LIN {X 0,Y 409.428,Z 527.797,A -85,B 0,C 180,E1 19478.338,E2 19478.338} C_VEL
LIN {X 0,Y 409.412,Z 527.774,A -85,B 0,C 180,E1 19474.343,E2 19474.343} C_VEL
LIN {X 0,Y 409.395,Z 527.8,A -85,B 0,C 180,E1 19470.531,E2 19470.531} C_VEL
LIN {X 0,Y 409.376,Z 527.779,A -85,B 0,C 180,E1 19466.862,E2 19466.862} C_VEL
LIN {X 0,Y 409.379,Z 527.798,A -85,B 0,C 180,E1 19462.967,E2 19462.967} C_VEL
LIN {X 0,Y 409.396,Z 527.782,A -85,B 0,C 180,E1 19459.251,E2 19459.251} C_VEL
LIN {X 0,Y 409.422,Z 527.785,A -85,B 0,C 180,E1 19455.438,E2 19455.438} C_VEL
LIN {X 0,Y 409.43,Z 527.788,A -85,B 0,C 180,E1 19451.552,E2 19451.552} C_VEL
LIN {X 0,Y 409.424,Z 527.77,A -85,B 0,C 180,E1 19447.578,E2 19447.578} C_VEL
LIN {X 0,Y 409.403,Z 527.799,A -85,B 0,C 180,E1 19443.781,E2 19443.781} C_VEL
LIN {X 0,Y 409.386,Z 527.767,A -85,B 0,C 180,E1 19440,E2 19440} C_VEL
LIN {X 0,Y 409.39,Z 527.799,A -85,B 0,C 180,E1 19436.079,E2 19436.079} C_VEL
LIN {X 0,Y 409.392,Z 527.773,A -85,B 0,C 180,E1 19432.139,E2 19432.139} C_VEL
LIN {X 0,Y 409.409,Z 527.797,A -85,B 0,C 180,E1 19428.305,E2 19428.305} C_VEL
LIN {X 0,Y 409.427,Z 527.78,A -85,B 0,C 180,E1 19424.417,E2 19424.417} C_VEL
LIN {X 0,Y 409.438,Z 527.787,A -85,B 0,C 180,E1 19420.488,E2 19420.488} C_VEL
LIN {X 0,Y 409.444,Z 527.796,A -85,B 0,C 180,E1 19416.544,E2 19416.544} C_VEL
LIN {X 0,Y 409.427,Z 527.783,A -85,B 0,C 180,E1 19412.67,E2 19412.67} C_VEL
LIN {X 0,Y 409.405,Z 527.789,A -85,B 0,C 180,E1 19408.982,E2 19408.982} C_VEL
LIN {X 0,Y 409.402,Z 527.793,A -85,B 0,C 180,E1 19405.14,E2 19405.14} C_VEL
LIN {X 0,Y 409.412,Z 527.79,A -85,B 0,C 180,E1 19401.303,E2 19401.303} C_VEL
LIN {X 0,Y 409.43,Z 527.79,A -85,B 0,C 180,E1 19397.516,E2 19397.516} C_VEL
LIN {X 0,Y 409.443,Z 527.799,A -85,B 0,C 180,E1 19393.711,E2 19393.711} C_VEL
LIN {X 0,Y 409.472,Z 528.088,A -85,B 0,C 180,E1 19392.071,E2 19392.071} C_VEL
LIN {X 0,Y 417.086,Z 549.044,A -85,B 0,C 180,E1 19388.821,E2 19388.821} C_VEL
LIN {X 0,Y 424.699,Z 571.518,A -85,B 0,C 180,E1 19385.686,E2 19385.686} C_VEL
LIN {X 0,Y 421.199,Z 607.599,A -85,B 0,C 180,E1 19382.122,E2 19382.122} C_VEL
LIN {X 0,Y 420.389,Z 616.971,A -85,B 0,C 180,E1 19381.23,E2 19381.23} C_VEL
LIN {X 0,Y 423.028,Z 641.822,A -85,B 0,C 180,E1 19380.601,E2 19380.601} C_VEL
LIN {X 0,Y 420.192,Z 815.687,A -85,B 0,C 180,E1 19377.631,E2 19377.631} C_VEL
LIN {X 0,Y 419.282,Z 834.324,A -85,B 0,C 180,E1 19377.076,E2 19377.076} C_VEL
LIN {X 0,Y 418.101,Z 852.187,A -85,B 0,C 180,E1 19376.296,E2 19376.296} C_VEL
LIN {X 0,Y 416.736,Z 869.515,A -85,B 0,C 180,E1 19375.281,E2 19375.281} C_VEL
LIN {X 0,Y 415.229,Z 886.464,A -85,B 0,C 180,E1 19374.013,E2 19374.013} C_VEL
LIN {X 0,Y 413.683,Z 902.434,A -85,B 0,C 180,E1 19372.525,E2 19372.525} C_VEL
LIN {X 0,Y 412.253,Z 917.439,A -85,B 0,C 180,E1 19370.813,E2 19370.813} C_VEL
LIN {X 0,Y 410.942,Z 931.411,A -85,B 0,C 180,E1 19368.881,E2 19368.881} C_VEL
LIN {X 0,Y 409.865,Z 944.229,A -85,B 0,C 180,E1 19366.73,E2 19366.73} C_VEL
LIN {X 0,Y 409.104,Z 955.381,A -85,B 0,C 180,E1 19364.436,E2 19364.436} C_VEL
LIN {X 0,Y 408.664,Z 964.433,A -85,B 0,C 180,E1 19362.147,E2 19362.147} C_VEL
LIN {X 0,Y 408.487,Z 972.044,A -85,B 0,C 180,E1 19359.724,E2 19359.724} C_VEL
LIN {X 0,Y 408.488,Z 977.818,A -85,B 0,C 180,E1 19357.314,E2 19357.314} C_VEL
LIN {X 0,Y 408.596,Z 981.892,A -85,B 0,C 180,E1 19354.915,E2 19354.915} C_VEL
LIN {X 0,Y 408.712,Z 984.339,A -85,B 0,C 180,E1 19352.525,E2 19352.525} C_VEL
LIN {X 0,Y 408.779,Z 985.198,A -85,B 0,C 180,E1 19350.002,E2 19350.002} C_VEL
LIN {X 0,Y 408.718,Z 984.298,A -85,B 0,C 180,E1 19347.478,E2 19347.478} C_VEL
LIN {X 0,Y 408.599,Z 981.642,A -85,B 0,C 180,E1 19344.948,E2 19344.948} C_VEL
LIN {X 0,Y 408.483,Z 977.183,A -85,B 0,C 180,E1 19342.407,E2 19342.407} C_VEL
LIN {X 0,Y 408.507,Z 970.81,A -85,B 0,C 180,E1 19339.853,E2 19339.853} C_VEL
LIN {X 0,Y 408.719,Z 962.882,A -85,B 0,C 180,E1 19337.428,E2 19337.428} C_VEL
LIN {X 0,Y 409.259,Z 952.866,A -85,B 0,C 180,E1 19334.994,E2 19334.994} C_VEL
LIN {X 0,Y 410.046,Z 942.036,A -85,B 0,C 180,E1 19332.843,E2 19332.843} C_VEL
LIN {X 0,Y 411.163,Z 929.405,A -85,B 0,C 180,E1 19330.766,E2 19330.766} C_VEL
LIN {X 0,Y 412.611,Z 914.663,A -85,B 0,C 180,E1 19328.764,E2 19328.764} C_VEL
LIN {X 0,Y 414.144,Z 899.377,A -85,B 0,C 180,E1 19327.055,E2 19327.055} C_VEL
LIN {X 0,Y 415.73,Z 883.929,A -85,B 0,C 180,E1 19325.644,E2 19325.644} C_VEL
LIN {X 0,Y 417.307,Z 866.913,A -85,B 0,C 180,E1 19324.388,E2 19324.388} C_VEL
LIN {X 0,Y 418.791,Z 849.197,A -85,B 0,C 180,E1 19323.373,E2 19323.373} C_VEL
LIN {X 0,Y 420.069,Z 830.603,A -85,B 0,C 180,E1 19322.594,E2 19322.594} C_VEL
LIN {X 0,Y 420.944,Z 811.694,A -85,B 0,C 180,E1 19322.072,E2 19322.072} C_VEL
LIN {X 0,Y 423.821,Z 639.08,A -85,B 0,C 180,E1 19319.074,E2 19319.074} C_VEL
LIN {X 0,Y 421.333,Z 617.013,A -85,B 0,C 180,E1 19318.434,E2 19318.434} C_VEL
LIN {X 0,Y 426.266,Z 573.613,A -85,B 0,C 180,E1 19314.039,E2 19314.039} C_VEL
LIN {X 0,Y 420.863,Z 557.04,A -85,B 0,C 180,E1 19311.511,E2 19311.511} C_VEL
LIN {X 0,Y 415.095,Z 541.83,A -85,B 0,C 180,E1 19308.89,E2 19308.89} C_VEL
LIN {X 0,Y 410.413,Z 530.778,A -85,B 0,C 180,E1 19306.755,E2 19306.755} C_VEL
LIN {X 0,Y 409.458,Z 527.95,A -85,B 0,C 180,E1 19306.13,E2 19306.13} C_VEL
LIN {X 0,Y 409.44,Z 527.788,A -85,B 0,C 180,E1 19302.187,E2 19302.187} C_VEL
LIN {X 0,Y 409.429,Z 527.787,A -85,B 0,C 180,E1 19298.337,E2 19298.337} C_VEL
LIN {X 0,Y 409.403,Z 527.796,A -85,B 0,C 180,E1 19294.513,E2 19294.513} C_VEL
LIN {X 0,Y 409.388,Z 527.799,A -85,B 0,C 180,E1 19290.693,E2 19290.693} C_VEL
LIN {X 0,Y 409.38,Z 527.798,A -85,B 0,C 180,E1 19286.862,E2 19286.862} C_VEL
LIN {X 0,Y 409.381,Z 527.791,A -85,B 0,C 180,E1 19282.977,E2 19282.977} C_VEL
LIN {X 0,Y 409.397,Z 527.783,A -85,B 0,C 180,E1 19279.251,E2 19279.251} C_VEL
LIN {X 0,Y 409.419,Z 527.784,A -85,B 0,C 180,E1 19275.438,E2 19275.438} C_VEL
LIN {X 0,Y 409.404,Z 527.801,A -85,B 0,C 180,E1 19271.552,E2 19271.552} C_VEL
LIN {X 0,Y 409.383,Z 527.799,A -85,B 0,C 180,E1 19267.72,E2 19267.72} C_VEL
LIN {X 0,Y 409.37,Z 527.787,A -85,B 0,C 180,E1 19263.921,E2 19263.921} C_VEL
LIN {X 0,Y 409.371,Z 527.786,A -85,B 0,C 180,E1 19260.14,E2 19260.14} C_VEL
LIN {X 0,Y 409.386,Z 527.796,A -85,B 0,C 180,E1 19256.359,E2 19256.359} C_VEL
LIN {X 0,Y 409.414,Z 527.799,A -85,B 0,C 180,E1 19252.563,E2 19252.563} C_VEL
LIN {X 0,Y 409.432,Z 527.798,A -85,B 0,C 180,E1 19248.734,E2 19248.734} C_VEL
LIN {X 0,Y 409.431,Z 527.795,A -85,B 0,C 180,E1 19244.852,E2 19244.852} C_VEL
LIN {X 0,Y 409.412,Z 527.798,A -85,B 0,C 180,E1 19241.046,E2 19241.046} C_VEL
LIN {X 0,Y 409.4,Z 527.803,A -85,B 0,C 180,E1 19237.301,E2 19237.301} C_VEL
LIN {X 0,Y 409.402,Z 527.794,A -85,B 0,C 180,E1 19233.349,E2 19233.349} C_VEL
LIN {X 0,Y 409.414,Z 527.839,A -85,B 0,C 180,E1 19229.471,E2 19229.471} C_VEL
LIN {X 0,Y 409.537,Z 528.542,A -85,B 0,C 180,E1 19229.156,E2 19229.156} C_VEL
LIN {X 0,Y 413.799,Z 540.293,A -85,B 0,C 180,E1 19226.404,E2 19226.404} C_VEL
LIN {X 0,Y 418.13,Z 554.109,A -85,B 0,C 180,E1 19223.453,E2 19223.453} C_VEL
LIN {X 0,Y 421.697,Z 567.85,A -85,B 0,C 180,E1 19220.767,E2 19220.767} C_VEL
LIN {X 0,Y 418.78,Z 594.647,A -85,B 0,C 180,E1 19216.728,E2 19216.728} C_VEL
LIN {X 0,Y 416.121,Z 622.884,A -85,B 0,C 180,E1 19212.555,E2 19212.555} C_VEL
LIN {X 0,Y 415.538,Z 630.261,A -85,B 0,C 180,E1 19211.502,E2 19211.502} C_VEL
LIN {X 0,Y 416.961,Z 637.693,A -85,B 0,C 180,E1 19211.191,E2 19211.191} C_VEL
LIN {X 0,Y 420.359,Z 656.969,A -85,B 0,C 180,E1 19210.559,E2 19210.559} C_VEL
LIN {X 0,Y 418.283,Z 753.864,A -85,B 0,C 180,E1 19208.726,E2 19208.726} C_VEL
LIN {X 0,Y 417.743,Z 769.981,A -85,B 0,C 180,E1 19208.156,E2 19208.156} C_VEL
LIN {X 0,Y 416.97,Z 784.418,A -85,B 0,C 180,E1 19207.391,E2 19207.391} C_VEL
LIN {X 0,Y 415.919,Z 799,A -85,B 0,C 180,E1 19206.335,E2 19206.335} C_VEL
LIN {X 0,Y 414.729,Z 811.961,A -85,B 0,C 180,E1 19205.094,E2 19205.094} C_VEL
LIN {X 0,Y 413.625,Z 823.119,A -85,B 0,C 180,E1 19203.741,E2 19203.741} C_VEL
LIN {X 0,Y 412.428,Z 833.983,A -85,B 0,C 180,E1 19202.063,E2 19202.063} C_VEL
LIN {X 0,Y 411.435,Z 842.658,A -85,B 0,C 180,E1 19200.358,E2 19200.358} C_VEL
LIN {X 0,Y 410.535,Z 850.51,A -85,B 0,C 180,E1 19198.35,E2 19198.35} C_VEL
LIN {X 0,Y 409.905,Z 856.206,A -85,B 0,C 180,E1 19196.351,E2 19196.351} C_VEL
LIN {X 0,Y 409.471,Z 860.386,A -85,B 0,C 180,E1 19194.215,E2 19194.215} C_VEL
LIN {X 0,Y 409.207,Z 862.789,A -85,B 0,C 180,E1 19191.949,E2 19191.949} C_VEL
LIN {X 0,Y 409.115,Z 863.297,A -85,B 0,C 180,E1 19189.792,E2 19189.792} C_VEL
LIN {X 0,Y 409.173,Z 861.968,A -85,B 0,C 180,E1 19187.488,E2 19187.488} C_VEL
LIN {X 0,Y 409.177,Z 861.878,A -85,B 0,C 180,E1 19187.409,E2 19187.409} C_VEL
LIN {X 0,Y 408.267,Z 860.683,A -85,B 0,C 180,E1 19186.342,E2 19186.342} C_VEL
LIN {X 0,Y 404.279,Z 858.032,A -85,B 0,C 180,E1 19184.487,E2 19184.487} C_VEL
LIN {X 0,Y 402.202,Z 855.385,A -85,B 0,C 180,E1 19183.225,E2 19183.225} C_VEL
LIN {X 0,Y 402.01,Z 853.771,A -85,B 0,C 180,E1 19182.633,E2 19182.633} C_VEL
LIN {X 0,Y 402.625,Z 847.266,A -85,B 0,C 180,E1 19180.731,E2 19180.731} C_VEL
LIN {X 0,Y 403.485,Z 838.789,A -85,B 0,C 180,E1 19178.835,E2 19178.835} C_VEL
LIN {X 0,Y 404.483,Z 828.762,A -85,B 0,C 180,E1 19177.097,E2 19177.097} C_VEL
LIN {X 0,Y 405.538,Z 817.784,A -85,B 0,C 180,E1 19175.587,E2 19175.587} C_VEL
LIN {X 0,Y 406.689,Z 804.448,A -85,B 0,C 180,E1 19174.157,E2 19174.157} C_VEL
LIN {X 0,Y 407.652,Z 791.603,A -85,B 0,C 180,E1 19173.091,E2 19173.091} C_VEL
LIN {X 0,Y 408.555,Z 776.319,A -85,B 0,C 180,E1 19172.137,E2 19172.137} C_VEL
LIN {X 0,Y 409.192,Z 760.052,A -85,B 0,C 180,E1 19171.446,E2 19171.446} C_VEL
LIN {X 0,Y 409.527,Z 743.398,A -85,B 0,C 180,E1 19171.032,E2 19171.032} C_VEL
LIN {X 0,Y 410.968,Z 654.967,A -85,B 0,C 180,E1 19169.399,E2 19169.399} C_VEL
LIN {X 0,Y 406.648,Z 630.171,A -85,B 0,C 180,E1 19168.625,E2 19168.625} C_VEL
LIN {X 0,Y 409.006,Z 601.035,A -85,B 0,C 180,E1 19164.387,E2 19164.387} C_VEL
LIN {X 0,Y 411.546,Z 573.669,A -85,B 0,C 180,E1 19160.349,E2 19160.349} C_VEL
LIN {X 0,Y 412.12,Z 566.266,A -85,B 0,C 180,E1 19159.232,E2 19159.232} C_VEL
LIN {X 0,Y 407.551,Z 549.156,A -85,B 0,C 180,E1 19156.088,E2 19156.088} C_VEL
LIN {X 0,Y 403.04,Z 533.934,A -85,B 0,C 180,E1 19153.127,E2 19153.127} C_VEL
LIN {X 0,Y 401.452,Z 528.917,A -85,B 0,C 180,E1 19152.068,E2 19152.068} C_VEL
LIN {X 0,Y 401.424,Z 528.776,A -85,B 0,C 180,E1 19148.215,E2 19148.215} C_VEL
LIN {X 0,Y 401.426,Z 528.779,A -85,B 0,C 180,E1 19144.317,E2 19144.317} C_VEL
LIN {X 0,Y 401.439,Z 528.746,A -85,B 0,C 180,E1 19140.616,E2 19140.616} C_VEL
LIN {X 0,Y 401.465,Z 528.773,A -85,B 0,C 180,E1 19136.777,E2 19136.777} C_VEL
LIN {X 0,Y 401.468,Z 528.774,A -85,B 0,C 180,E1 19132.842,E2 19132.842} C_VEL
LIN {X 0,Y 401.455,Z 528.785,A -85,B 0,C 180,E1 19128.995,E2 19128.995} C_VEL
LIN {X 0,Y 401.437,Z 528.788,A -85,B 0,C 180,E1 19125.184,E2 19125.184} C_VEL
LIN {X 0,Y 401.428,Z 528.769,A -85,B 0,C 180,E1 19121.304,E2 19121.304} C_VEL
LIN {X 0,Y 401.433,Z 528.791,A -85,B 0,C 180,E1 19117.392,E2 19117.392} C_VEL
LIN {X 0,Y 401.437,Z 528.767,A -85,B 0,C 180,E1 19113.453,E2 19113.453} C_VEL
LIN {X 0,Y 401.456,Z 528.788,A -85,B 0,C 180,E1 19109.638,E2 19109.638} C_VEL
LIN {X 0,Y 401.478,Z 528.757,A -85,B 0,C 180,E1 19105.838,E2 19105.838} C_VEL
LIN {X 0,Y 401.492,Z 528.789,A -85,B 0,C 180,E1 19101.935,E2 19101.935} C_VEL
LIN {X 0,Y 401.474,Z 528.755,A -85,B 0,C 180,E1 19097.953,E2 19097.953} C_VEL
LIN {X 0,Y 401.457,Z 528.785,A -85,B 0,C 180,E1 19094.128,E2 19094.128} C_VEL
LIN {X 0,Y 401.444,Z 528.772,A -85,B 0,C 180,E1 19090.331,E2 19090.331} C_VEL
LIN {X 0,Y 401.446,Z 528.779,A -85,B 0,C 180,E1 19086.43,E2 19086.43} C_VEL
LIN {X 0,Y 401.454,Z 528.777,A -85,B 0,C 180,E1 19082.57,E2 19082.57} C_VEL
LIN {X 0,Y 401.472,Z 528.771,A -85,B 0,C 180,E1 19078.716,E2 19078.716} C_VEL
LIN {X 0,Y 401.491,Z 528.778,A -85,B 0,C 180,E1 19074.857,E2 19074.857} C_VEL
LIN {X 0,Y 401.495,Z 528.766,A -85,B 0,C 180,E1 19070.974,E2 19070.974} C_VEL
LIN {X 0,Y 401.484,Z 528.778,A -85,B 0,C 180,E1 19067.048,E2 19067.048} C_VEL
LIN {X 0,Y 401.471,Z 528.781,A -85,B 0,C 180,E1 19063.208,E2 19063.208} C_VEL
LIN {X 0,Y 401.458,Z 528.773,A -85,B 0,C 180,E1 19059.441,E2 19059.441} C_VEL
LIN {X 0,Y 401.462,Z 528.788,A -85,B 0,C 180,E1 19055.423,E2 19055.423} C_VEL
LIN {X 0,Y 401.463,Z 528.787,A -85,B 0,C 180,E1 19051.433,E2 19051.433} C_VEL
LIN {X 0,Y 401.476,Z 528.783,A -85,B 0,C 180,E1 19047.589,E2 19047.589} C_VEL
LIN {X 0,Y 401.486,Z 528.781,A -85,B 0,C 180,E1 19043.65,E2 19043.65} C_VEL
LIN {X 0,Y 401.511,Z 528.782,A -85,B 0,C 180,E1 19039.837,E2 19039.837} C_VEL
LIN {X 0,Y 401.503,Z 528.78,A -85,B 0,C 180,E1 19035.791,E2 19035.791} C_VEL
LIN {X 0,Y 401.506,Z 529.047,A -85,B 0,C 180,E1 19032.805,E2 19032.805} C_VEL
LIN {X 0,Y 408.035,Z 546.843,A -85,B 0,C 180,E1 19029.917,E2 19029.917} C_VEL
LIN {X 0,Y 415.804,Z 569.544,A -85,B 0,C 180,E1 19026.607,E2 19026.607} C_VEL
LIN {X 0,Y 417.398,Z 574.481,A -85,B 0,C 180,E1 19025.935,E2 19025.935} C_VEL
LIN {X 0,Y 413.013,Z 617.101,A -85,B 0,C 180,E1 19021.69,E2 19021.69} C_VEL
LIN {X 0,Y 415.688,Z 642.766,A -85,B 0,C 180,E1 19021.026,E2 19021.026} C_VEL
LIN {X 0,Y 412.724,Z 815.114,A -85,B 0,C 180,E1 19018.032,E2 19018.032} C_VEL
LIN {X 0,Y 411.776,Z 833.715,A -85,B 0,C 180,E1 19017.469,E2 19017.469} C_VEL
LIN {X 0,Y 410.528,Z 851.793,A -85,B 0,C 180,E1 19016.663,E2 19016.663} C_VEL
LIN {X 0,Y 409.033,Z 869.817,A -85,B 0,C 180,E1 19015.578,E2 19015.578} C_VEL
LIN {X 0,Y 407.45,Z 886.751,A -85,B 0,C 180,E1 19014.27,E2 19014.27} C_VEL
LIN {X 0,Y 405.85,Z 902.538,A -85,B 0,C 180,E1 19012.755,E2 19012.755} C_VEL
LIN {X 0,Y 404.369,Z 917.411,A -85,B 0,C 180,E1 19011.01,E2 19011.01} C_VEL
LIN {X 0,Y 403.019,Z 931.196,A -85,B 0,C 180,E1 19009.051,E2 19009.051} C_VEL
LIN {X 0,Y 401.931,Z 943.503,A -85,B 0,C 180,E1 19006.921,E2 19006.921} C_VEL
LIN {X 0,Y 401.141,Z 954.588,A -85,B 0,C 180,E1 19004.581,E2 19004.581} C_VEL
LIN {X 0,Y 400.692,Z 963.579,A -85,B 0,C 180,E1 19002.246,E2 19002.246} C_VEL
LIN {X 0,Y 400.522,Z 971.13,A -85,B 0,C 180,E1 18999.774,E2 18999.774} C_VEL
LIN {X 0,Y 400.542,Z 976.841,A -85,B 0,C 180,E1 18997.315,E2 18997.315} C_VEL
LIN {X 0,Y 400.671,Z 980.848,A -85,B 0,C 180,E1 18994.868,E2 18994.868} C_VEL
LIN {X 0,Y 400.801,Z 983.229,A -85,B 0,C 180,E1 18992.432,E2 18992.432} C_VEL
LIN {X 0,Y 400.862,Z 984.008,A -85,B 0,C 180,E1 18989.859,E2 18989.859} C_VEL
LIN {X 0,Y 400.791,Z 983.021,A -85,B 0,C 180,E1 18987.285,E2 18987.285} C_VEL
LIN {X 0,Y 400.647,Z 980.262,A -85,B 0,C 180,E1 18984.704,E2 18984.704} C_VEL
LIN {X 0,Y 400.517,Z 975.677,A -85,B 0,C 180,E1 18982.111,E2 18982.111} C_VEL
LIN {X 0,Y 400.54,Z 969.412,A -85,B 0,C 180,E1 18979.587,E2 18979.587} C_VEL
LIN {X 0,Y 400.762,Z 961.642,A -85,B 0,C 180,E1 18977.174,E2 18977.174} C_VEL
LIN {X 0,Y 401.3,Z 952.266,A -85,B 0,C 180,E1 18974.837,E2 18974.837} C_VEL
LIN {X 0,Y 402.19,Z 940.755,A -85,B 0,C 180,E1 18972.497,E2 18972.497} C_VEL
LIN {X 0,Y 403.402,Z 928.028,A -85,B 0,C 180,E1 18970.365,E2 18970.365} C_VEL
LIN {X 0,Y 404.937,Z 913.359,A -85,B 0,C 180,E1 18968.341,E2 18968.341} C_VEL
LIN {X 0,Y 406.577,Z 898.013,A -85,B 0,C 180,E1 18966.603,E2 18966.603} C_VEL
LIN {X 0,Y 408.361,Z 881.645,A -85,B 0,C 180,E1 18965.098,E2 18965.098} C_VEL
LIN {X 0,Y 410.061,Z 864.155,A -85,B 0,C 180,E1 18963.815,E2 18963.815} C_VEL
LIN {X 0,Y 411.562,Z 846.627,A -85,B 0,C 180,E1 18962.828,E2 18962.828} C_VEL
LIN {X 0,Y 412.867,Z 828.371,A -85,B 0,C 180,E1 18962.08,E2 18962.08} C_VEL
LIN {X 0,Y 413.719,Z 809.659,A -85,B 0,C 180,E1 18961.574,E2 18961.574} C_VEL
LIN {X 0,Y 416.751,Z 639.969,A -85,B 0,C 180,E1 18958.57,E2 18958.57} C_VEL
LIN {X 0,Y 414.205,Z 617.187,A -85,B 0,C 180,E1 18957.891,E2 18957.891} C_VEL
LIN {X 0,Y 419.131,Z 576.561,A -85,B 0,C 180,E1 18953.692,E2 18953.692} C_VEL
LIN {X 0,Y 414.105,Z 560.904,A -85,B 0,C 180,E1 18951.25,E2 18951.25} C_VEL
LIN {X 0,Y 408.565,Z 546.162,A -85,B 0,C 180,E1 18948.649,E2 18948.649} C_VEL
LIN {X 0,Y 403.106,Z 532.757,A -85,B 0,C 180,E1 18945.998,E2 18945.998} C_VEL
LIN {X 0,Y 401.502,Z 529.061,A -85,B 0,C 180,E1 18945.161,E2 18945.161} C_VEL
LIN {X 0,Y 401.499,Z 528.776,A -85,B 0,C 180,E1 18942.059,E2 18942.059} C_VEL
LIN {X 0,Y 401.501,Z 528.776,A -85,B 0,C 180,E1 18938.109,E2 18938.109} C_VEL
LIN {X 0,Y 401.492,Z 528.785,A -85,B 0,C 180,E1 18934.078,E2 18934.078} C_VEL
LIN {X 0,Y 401.492,Z 528.787,A -85,B 0,C 180,E1 18930.037,E2 18930.037} C_VEL
LIN {X 0,Y 401.464,Z 528.788,A -85,B 0,C 180,E1 18926.156,E2 18926.156} C_VEL
LIN {X 0,Y 401.44,Z 528.787,A -85,B 0,C 180,E1 18922.4,E2 18922.4} C_VEL
LIN {X 0,Y 401.431,Z 528.777,A -85,B 0,C 180,E1 18918.591,E2 18918.591} C_VEL
LIN {X 0,Y 401.428,Z 528.772,A -85,B 0,C 180,E1 18914.717,E2 18914.717} C_VEL
LIN {X 0,Y 401.441,Z 528.784,A -85,B 0,C 180,E1 18910.911,E2 18910.911} C_VEL
LIN {X 0,Y 401.462,Z 528.791,A -85,B 0,C 180,E1 18907.009,E2 18907.009} C_VEL
LIN {X 0,Y 401.475,Z 528.78,A -85,B 0,C 180,E1 18903.077,E2 18903.077} C_VEL
LIN {X 0,Y 401.484,Z 528.769,A -85,B 0,C 180,E1 18899.144,E2 18899.144} C_VEL
LIN {X 0,Y 401.475,Z 528.77,A -85,B 0,C 180,E1 18895.142,E2 18895.142} C_VEL
LIN {X 0,Y 401.458,Z 528.778,A -85,B 0,C 180,E1 18891.355,E2 18891.355} C_VEL
LIN {X 0,Y 401.454,Z 528.784,A -85,B 0,C 180,E1 18887.474,E2 18887.474} C_VEL
LIN {X 0,Y 401.454,Z 528.788,A -85,B 0,C 180,E1 18883.654,E2 18883.654} C_VEL
LIN {X 0,Y 401.462,Z 528.783,A -85,B 0,C 180,E1 18879.745,E2 18879.745} C_VEL
LIN {X 0,Y 401.474,Z 528.777,A -85,B 0,C 180,E1 18875.893,E2 18875.893} C_VEL
LIN {X 0,Y 401.502,Z 528.78,A -85,B 0,C 180,E1 18872.084,E2 18872.084} C_VEL
LIN {X 0,Y 401.552,Z 529.069,A -85,B 0,C 180,E1 18870.255,E2 18870.255} C_VEL
LIN {X 0,Y 406.238,Z 542.209,A -85,B 0,C 180,E1 18867.047,E2 18867.047} C_VEL
LIN {X 0,Y 410.785,Z 556.507,A -85,B 0,C 180,E1 18863.9,E2 18863.9} C_VEL
LIN {X 0,Y 414.447,Z 570.745,A -85,B 0,C 180,E1 18861.038,E2 18861.038} C_VEL
LIN {X 0,Y 411.346,Z 597.73,A -85,B 0,C 180,E1 18856.919,E2 18856.919} C_VEL
LIN {X 0,Y 408.536,Z 625.969,A -85,B 0,C 180,E1 18852.675,E2 18852.675} C_VEL
LIN {X 0,Y 408.22,Z 630.135,A -85,B 0,C 180,E1 18852.085,E2 18852.085} C_VEL
LIN {X 0,Y 409.952,Z 639.021,A -85,B 0,C 180,E1 18851.713,E2 18851.713} C_VEL
LIN {X 0,Y 413.308,Z 658.122,A -85,B 0,C 180,E1 18851.067,E2 18851.067} C_VEL
LIN {X 0,Y 411.119,Z 754.468,A -85,B 0,C 180,E1 18849.211,E2 18849.211} C_VEL
LIN {X 0,Y 410.547,Z 770.607,A -85,B 0,C 180,E1 18848.632,E2 18848.632} C_VEL
LIN {X 0,Y 409.724,Z 785.076,A -85,B 0,C 180,E1 18847.854,E2 18847.854} C_VEL
LIN {X 0,Y 408.645,Z 799.137,A -85,B 0,C 180,E1 18846.825,E2 18846.825} C_VEL
LIN {X 0,Y 407.452,Z 811.541,A -85,B 0,C 180,E1 18845.643,E2 18845.643} C_VEL
LIN {X 0,Y 406.142,Z 823.891,A -85,B 0,C 180,E1 18844.14,E2 18844.14} C_VEL
LIN {X 0,Y 404.832,Z 834.961,A -85,B 0,C 180,E1 18842.403,E2 18842.403} C_VEL
LIN {X 0,Y 403.764,Z 843.664,A -85,B 0,C 180,E1 18840.667,E2 18840.667} C_VEL
LIN {X 0,Y 402.785,Z 851.537,A -85,B 0,C 180,E1 18838.622,E2 18838.622} C_VEL
LIN {X 0,Y 402.093,Z 857.273,A -85,B 0,C 180,E1 18836.585,E2 18836.585} C_VEL
LIN {X 0,Y 401.612,Z 861.494,A -85,B 0,C 180,E1 18834.407,E2 18834.407} C_VEL
LIN {X 0,Y 401.312,Z 863.933,A -85,B 0,C 180,E1 18832.095,E2 18832.095} C_VEL
LIN {X 0,Y 401.207,Z 864.512,A -85,B 0,C 180,E1 18829.96,E2 18829.96} C_VEL
LIN {X 0,Y 401.257,Z 863.218,A -85,B 0,C 180,E1 18827.545,E2 18827.545} C_VEL
LIN {X 0,Y 401.474,Z 860.086,A -85,B 0,C 180,E1 18825.304,E2 18825.304} C_VEL
LIN {X 0,Y 401.863,Z 855.46,A -85,B 0,C 180,E1 18823.229,E2 18823.229} C_VEL
LIN {X 0,Y 402.01,Z 853.771,A -85,B 0,C 180,E1 18822.633,E2 18822.633} C_VEL
LIN {X 0,Y 401.342,Z 850.78,A -85,B 0,C 180,E1 18821.614,E2 18821.614} C_VEL
LIN {X 0,Y 397.654,Z 844.742,A -85,B 0,C 180,E1 18819.79,E2 18819.79} C_VEL
LIN {X 0,Y 396.013,Z 840.237,A -85,B 0,C 180,E1 18818.704,E2 18818.704} C_VEL
LIN {X 0,Y 395.947,Z 837.653,A -85,B 0,C 180,E1 18818.182,E2 18818.182} C_VEL
LIN {X 0,Y 397.049,Z 827.221,A -85,B 0,C 180,E1 18816.432,E2 18816.432} C_VEL
LIN {X 0,Y 398.248,Z 814.92,A -85,B 0,C 180,E1 18814.822,E2 18814.822} C_VEL
LIN {X 0,Y 399.383,Z 802.062,A -85,B 0,C 180,E1 18813.514,E2 18813.514} C_VEL
LIN {X 0,Y 400.407,Z 788.323,A -85,B 0,C 180,E1 18812.431,E2 18812.431} C_VEL
LIN {X 0,Y 401.282,Z 772.699,A -85,B 0,C 180,E1 18811.533,E2 18811.533} C_VEL
LIN {X 0,Y 401.837,Z 757.365,A -85,B 0,C 180,E1 18810.938,E2 18810.938} C_VEL
LIN {X 0,Y 402.302,Z 733.276,A -85,B 0,C 180,E1 18810.414,E2 18810.414} C_VEL
LIN {X 0,Y 403.614,Z 656.089,A -85,B 0,C 180,E1 18808.969,E2 18808.969} C_VEL
LIN {X 0,Y 399.105,Z 630.293,A -85,B 0,C 180,E1 18808.164,E2 18808.164} C_VEL
LIN {X 0,Y 401.592,Z 601.019,A -85,B 0,C 180,E1 18803.853,E2 18803.853} C_VEL
LIN {X 0,Y 404.307,Z 573.606,A -85,B 0,C 180,E1 18799.743,E2 18799.743} C_VEL
LIN {X 0,Y 404.695,Z 568.962,A -85,B 0,C 180,E1 18799.032,E2 18799.032} C_VEL
LIN {X 0,Y 400.139,Z 551.785,A -85,B 0,C 180,E1 18795.821,E2 18795.821} C_VEL
LIN {X 0,Y 395.189,Z 535.216,A -85,B 0,C 180,E1 18792.525,E2 18792.525} C_VEL
LIN {X 0,Y 393.553,Z 529.9,A -85,B 0,C 180,E1 18791.379,E2 18791.379} C_VEL
LIN {X 0,Y 393.537,Z 529.737,A -85,B 0,C 180,E1 18787.283,E2 18787.283} C_VEL
LIN {X 0,Y 393.525,Z 529.779,A -85,B 0,C 180,E1 18783.275,E2 18783.275} C_VEL
LIN {X 0,Y 393.494,Z 529.723,A -85,B 0,C 180,E1 18779.457,E2 18779.457} C_VEL
LIN {X 0,Y 393.488,Z 529.781,A -85,B 0,C 180,E1 18775.661,E2 18775.661} C_VEL
LIN {X 0,Y 393.486,Z 529.775,A -85,B 0,C 180,E1 18771.685,E2 18771.685} C_VEL
LIN {X 0,Y 393.486,Z 529.762,A -85,B 0,C 180,E1 18767.674,E2 18767.674} C_VEL
LIN {X 0,Y 393.494,Z 529.779,A -85,B 0,C 180,E1 18763.721,E2 18763.721} C_VEL
LIN {X 0,Y 393.504,Z 529.767,A -85,B 0,C 180,E1 18759.815,E2 18759.815} C_VEL
LIN {X 0,Y 393.534,Z 529.767,A -85,B 0,C 180,E1 18756.108,E2 18756.108} C_VEL
LIN {X 0,Y 393.543,Z 529.763,A -85,B 0,C 180,E1 18752.073,E2 18752.073} C_VEL
LIN {X 0,Y 393.543,Z 529.762,A -85,B 0,C 180,E1 18748.169,E2 18748.169} C_VEL
LIN {X 0,Y 393.534,Z 529.76,A -85,B 0,C 180,E1 18744.146,E2 18744.146} C_VEL
LIN {X 0,Y 393.514,Z 529.775,A -85,B 0,C 180,E1 18740.36,E2 18740.36} C_VEL
LIN {X 0,Y 393.501,Z 529.753,A -85,B 0,C 180,E1 18736.534,E2 18736.534} C_VEL
LIN {X 0,Y 393.505,Z 529.777,A -85,B 0,C 180,E1 18732.622,E2 18732.622} C_VEL
LIN {X 0,Y 393.506,Z 529.741,A -85,B 0,C 180,E1 18728.622,E2 18728.622} C_VEL
LIN {X 0,Y 393.524,Z 529.775,A -85,B 0,C 180,E1 18724.81,E2 18724.81} C_VEL
LIN {X 0,Y 393.536,Z 529.74,A -85,B 0,C 180,E1 18720.874,E2 18720.874} C_VEL
LIN {X 0,Y 393.552,Z 529.776,A -85,B 0,C 180,E1 18716.942,E2 18716.942} C_VEL
LIN {X 0,Y 393.563,Z 529.745,A -85,B 0,C 180,E1 18712.996,E2 18712.996} C_VEL
LIN {X 0,Y 393.552,Z 529.776,A -85,B 0,C 180,E1 18709.016,E2 18709.016} C_VEL
LIN {X 0,Y 393.537,Z 529.752,A -85,B 0,C 180,E1 18705.131,E2 18705.131} C_VEL
LIN {X 0,Y 393.531,Z 529.779,A -85,B 0,C 180,E1 18701.176,E2 18701.176} C_VEL
LIN {X 0,Y 393.521,Z 529.771,A -85,B 0,C 180,E1 18697.259,E2 18697.259} C_VEL
LIN {X 0,Y 393.523,Z 529.759,A -85,B 0,C 180,E1 18693.275,E2 18693.275} C_VEL
LIN {X 0,Y 393.525,Z 529.768,A -85,B 0,C 180,E1 18689.29,E2 18689.29} C_VEL
LIN {X 0,Y 393.527,Z 529.771,A -85,B 0,C 180,E1 18685.311,E2 18685.311} C_VEL
LIN {X 0,Y 393.535,Z 529.767,A -85,B 0,C 180,E1 18681.317,E2 18681.317} C_VEL
LIN {X 0,Y 393.549,Z 529.768,A -85,B 0,C 180,E1 18677.455,E2 18677.455} C_VEL
LIN {X 0,Y 393.589,Z 529.973,A -85,B 0,C 180,E1 18673.55,E2 18673.55} C_VEL
LIN {X 0,Y 401.018,Z 550.323,A -85,B 0,C 180,E1 18670.165,E2 18670.165} C_VEL
LIN {X 0,Y 408.607,Z 572.641,A -85,B 0,C 180,E1 18666.854,E2 18666.854} C_VEL
LIN {X 0,Y 409.99,Z 576.832,A -85,B 0,C 180,E1 18666.263,E2 18666.263} C_VEL
LIN {X 0,Y 405.638,Z 617.026,A -85,B 0,C 180,E1 18662.168,E2 18662.168} C_VEL
LIN {X 0,Y 408.367,Z 643.803,A -85,B 0,C 180,E1 18661.464,E2 18661.464} C_VEL
LIN {X 0,Y 405.274,Z 814.539,A -85,B 0,C 180,E1 18658.449,E2 18658.449} C_VEL
LIN {X 0,Y 404.296,Z 833.064,A -85,B 0,C 180,E1 18657.878,E2 18657.878} C_VEL
LIN {X 0,Y 403.03,Z 850.733,A -85,B 0,C 180,E1 18657.079,E2 18657.079} C_VEL
LIN {X 0,Y 401.483,Z 868.542,A -85,B 0,C 180,E1 18655.996,E2 18655.996} C_VEL
LIN {X 0,Y 399.854,Z 885.346,A -85,B 0,C 180,E1 18654.682,E2 18654.682} C_VEL
LIN {X 0,Y 398.165,Z 901.215,A -85,B 0,C 180,E1 18653.141,E2 18653.141} C_VEL
LIN {X 0,Y 396.604,Z 916.148,A -85,B 0,C 180,E1 18651.364,E2 18651.364} C_VEL
LIN {X 0,Y 395.177,Z 930.043,A -85,B 0,C 180,E1 18649.357,E2 18649.357} C_VEL
LIN {X 0,Y 394.001,Z 942.727,A -85,B 0,C 180,E1 18647.12,E2 18647.12} C_VEL
LIN {X 0,Y 393.181,Z 953.784,A -85,B 0,C 180,E1 18644.733,E2 18644.733} C_VEL
LIN {X 0,Y 392.72,Z 962.723,A -85,B 0,C 180,E1 18642.35,E2 18642.35} C_VEL
LIN {X 0,Y 392.558,Z 970.214,A -85,B 0,C 180,E1 18639.827,E2 18639.827} C_VEL
LIN {X 0,Y 392.596,Z 975.863,A -85,B 0,C 180,E1 18637.317,E2 18637.317} C_VEL
LIN {X 0,Y 392.747,Z 979.803,A -85,B 0,C 180,E1 18634.821,E2 18634.821} C_VEL
LIN {X 0,Y 392.892,Z 982.109,A -85,B 0,C 180,E1 18632.335,E2 18632.335} C_VEL
LIN {X 0,Y 392.949,Z 982.829,A -85,B 0,C 180,E1 18629.856,E2 18629.856} C_VEL
LIN {X 0,Y 392.869,Z 981.845,A -85,B 0,C 180,E1 18627.23,E2 18627.23} C_VEL
LIN {X 0,Y 392.7,Z 979.08,A -85,B 0,C 180,E1 18624.597,E2 18624.597} C_VEL
LIN {X 0,Y 392.556,Z 974.482,A -85,B 0,C 180,E1 18621.95,E2 18621.95} C_VEL
LIN {X 0,Y 392.568,Z 968.38,A -85,B 0,C 180,E1 18619.436,E2 18619.436} C_VEL
LIN {X 0,Y 392.813,Z 960.421,A -85,B 0,C 180,E1 18616.91,E2 18616.91} C_VEL
LIN {X 0,Y 393.425,Z 950.522,A -85,B 0,C 180,E1 18614.407,E2 18614.407} C_VEL
LIN {X 0,Y 394.348,Z 939.525,A -85,B 0,C 180,E1 18612.137,E2 18612.137} C_VEL
LIN {X 0,Y 395.589,Z 927.341,A -85,B 0,C 180,E1 18610.053,E2 18610.053} C_VEL
LIN {X 0,Y 397.158,Z 913.206,A -85,B 0,C 180,E1 18608.05,E2 18608.05} C_VEL
LIN {X 0,Y 398.879,Z 898.031,A -85,B 0,C 180,E1 18606.281,E2 18606.281} C_VEL
LIN {X 0,Y 400.743,Z 881.871,A -85,B 0,C 180,E1 18604.749,E2 18604.749} C_VEL
LIN {X 0,Y 402.525,Z 864.753,A -85,B 0,C 180,E1 18603.446,E2 18603.446} C_VEL
LIN {X 0,Y 404.159,Z 847.129,A -85,B 0,C 180,E1 18602.408,E2 18602.408} C_VEL
LIN {X 0,Y 405.589,Z 828.498,A -85,B 0,C 180,E1 18601.615,E2 18601.615} C_VEL
LIN {X 0,Y 406.506,Z 809.925,A -85,B 0,C 180,E1 18601.091,E2 18601.091} C_VEL
LIN {X 0,Y 409.726,Z 640.883,A -85,B 0,C 180,E1 18598.047,E2 18598.047} C_VEL
LIN {X 0,Y 407.123,Z 617.318,A -85,B 0,C 180,E1 18597.324,E2 18597.324} C_VEL
LIN {X 0,Y 411.959,Z 579.169,A -85,B 0,C 180,E1 18593.286,E2 18593.286} C_VEL
LIN {X 0,Y 406.658,Z 562.717,A -85,B 0,C 180,E1 18590.635,E2 18590.635} C_VEL
LIN {X 0,Y 400.847,Z 547.365,A -85,B 0,C 180,E1 18587.802,E2 18587.802} C_VEL
LIN {X 0,Y 394.957,Z 533.455,A -85,B 0,C 180,E1 18584.867,E2 18584.867} C_VEL
LIN {X 0,Y 393.576,Z 529.939,A -85,B 0,C 180,E1 18584.01,E2 18584.01} C_VEL
LIN {X 0,Y 393.568,Z 529.773,A -85,B 0,C 180,E1 18580.129,E2 18580.129} C_VEL
LIN {X 0,Y 393.55,Z 529.765,A -85,B 0,C 180,E1 18576.116,E2 18576.116} C_VEL
LIN {X 0,Y 393.539,Z 529.763,A -85,B 0,C 180,E1 18572.227,E2 18572.227} C_VEL
LIN {X 0,Y 393.514,Z 529.766,A -85,B 0,C 180,E1 18568.475,E2 18568.475} C_VEL
LIN {X 0,Y 393.5,Z 529.769,A -85,B 0,C 180,E1 18564.557,E2 18564.557} C_VEL
LIN {X 0,Y 393.495,Z 529.779,A -85,B 0,C 180,E1 18560.683,E2 18560.683} C_VEL
LIN {X 0,Y 393.493,Z 529.782,A -85,B 0,C 180,E1 18556.686,E2 18556.686} C_VEL
LIN {X 0,Y 393.494,Z 529.779,A -85,B 0,C 180,E1 18552.771,E2 18552.771} C_VEL
LIN {X 0,Y 393.506,Z 529.763,A -85,B 0,C 180,E1 18548.916,E2 18548.916} C_VEL
LIN {X 0,Y 393.532,Z 529.757,A -85,B 0,C 180,E1 18545.102,E2 18545.102} C_VEL
LIN {X 0,Y 393.544,Z 529.765,A -85,B 0,C 180,E1 18541.019,E2 18541.019} C_VEL
LIN {X 0,Y 393.541,Z 529.777,A -85,B 0,C 180,E1 18537.087,E2 18537.087} C_VEL
LIN {X 0,Y 393.552,Z 529.776,A -85,B 0,C 180,E1 18532.995,E2 18532.995} C_VEL
LIN {X 0,Y 393.542,Z 529.772,A -85,B 0,C 180,E1 18529.015,E2 18529.015} C_VEL
LIN {X 0,Y 393.53,Z 529.771,A -85,B 0,C 180,E1 18525.13,E2 18525.13} C_VEL
LIN {X 0,Y 393.527,Z 529.776,A -85,B 0,C 180,E1 18521.175,E2 18521.175} C_VEL
LIN {X 0,Y 393.524,Z 529.781,A -85,B 0,C 180,E1 18517.249,E2 18517.249} C_VEL
LIN {X 0,Y 393.526,Z 529.77,A -85,B 0,C 180,E1 18513.274,E2 18513.274} C_VEL
LIN {X 0,Y 393.573,Z 530.09,A -85,B 0,C 180,E1 18511.317,E2 18511.317} C_VEL
LIN {X 0,Y 398.236,Z 542.653,A -85,B 0,C 180,E1 18508.086,E2 18508.086} C_VEL
LIN {X 0,Y 402.582,Z 556.068,A -85,B 0,C 180,E1 18504.99,E2 18504.99} C_VEL
LIN {X 0,Y 406.254,Z 569.399,A -85,B 0,C 180,E1 18502.179,E2 18502.179} C_VEL
LIN {X 0,Y 407.159,Z 574.319,A -85,B 0,C 180,E1 18501.229,E2 18501.229} C_VEL
LIN {X 0,Y 403.897,Z 600.966,A -85,B 0,C 180,E1 18497.096,E2 18497.096} C_VEL
LIN {X 0,Y 400.996,Z 628.738,A -85,B 0,C 180,E1 18492.855,E2 18492.855} C_VEL
LIN {X 0,Y 400.991,Z 630.643,A -85,B 0,C 180,E1 18492.644,E2 18492.644} C_VEL
LIN {X 0,Y 406.308,Z 658.578,A -85,B 0,C 180,E1 18491.605,E2 18491.605} C_VEL
LIN {X 0,Y 403.986,Z 755.036,A -85,B 0,C 180,E1 18489.715,E2 18489.715} C_VEL
LIN {X 0,Y 403.386,Z 771.085,A -85,B 0,C 180,E1 18489.132,E2 18489.132} C_VEL
LIN {X 0,Y 402.561,Z 785.093,A -85,B 0,C 180,E1 18488.378,E2 18488.378} C_VEL
LIN {X 0,Y 401.326,Z 800.291,A -85,B 0,C 180,E1 18487.252,E2 18487.252} C_VEL
LIN {X 0,Y 399.981,Z 813.357,A -85,B 0,C 180,E1 18485.97,E2 18485.97} C_VEL
LIN {X 0,Y 398.666,Z 824.96,A -85,B 0,C 180,E1 18484.523,E2 18484.523} C_VEL
LIN {X 0,Y 397.265,Z 836.023,A -85,B 0,C 180,E1 18482.755,E2 18482.755} C_VEL
LIN {X 0,Y 396.115,Z 844.717,A -85,B 0,C 180,E1 18480.988,E2 18480.988} C_VEL
LIN {X 0,Y 395.032,Z 852.721,A -85,B 0,C 180,E1 18478.865,E2 18478.865} C_VEL
LIN {X 0,Y 394.279,Z 858.43,A -85,B 0,C 180,E1 18476.792,E2 18476.792} C_VEL
LIN {X 0,Y 393.757,Z 862.595,A -85,B 0,C 180,E1 18474.606,E2 18474.606} C_VEL
LIN {X 0,Y 393.428,Z 865.028,A -85,B 0,C 180,E1 18472.32,E2 18472.32} C_VEL
LIN {X 0,Y 393.299,Z 865.713,A -85,B 0,C 180,E1 18470.068,E2 18470.068} C_VEL
LIN {X 0,Y 393.339,Z 864.46,A -85,B 0,C 180,E1 18467.604,E2 18467.604} C_VEL
LIN {X 0,Y 393.543,Z 861.669,A -85,B 0,C 180,E1 18465.469,E2 18465.469} C_VEL
LIN {X 0,Y 393.968,Z 856.853,A -85,B 0,C 180,E1 18463.201,E2 18463.201} C_VEL
LIN {X 0,Y 394.588,Z 850.407,A -85,B 0,C 180,E1 18461.101,E2 18461.101} C_VEL
LIN {X 0,Y 395.426,Z 842.541,A -85,B 0,C 180,E1 18459.164,E2 18459.164} C_VEL
LIN {X 0,Y 395.947,Z 837.653,A -85,B 0,C 180,E1 18458.182,E2 18458.182} C_VEL
LIN {X 0,Y 395.501,Z 832.965,A -85,B 0,C 180,E1 18457.286,E2 18457.286} C_VEL
LIN {X 0,Y 392.213,Z 824.091,A -85,B 0,C 180,E1 18455.677,E2 18455.677} C_VEL
LIN {X 0,Y 390.756,Z 817.925,A -85,B 0,C 180,E1 18454.761,E2 18454.761} C_VEL
LIN {X 0,Y 390.744,Z 814.515,A -85,B 0,C 180,E1 18454.346,E2 18454.346} C_VEL
LIN {X 0,Y 391.972,Z 801.072,A -85,B 0,C 180,E1 18452.995,E2 18452.995} C_VEL
LIN {X 0,Y 392.972,Z 787.787,A -85,B 0,C 180,E1 18451.966,E2 18451.966} C_VEL
LIN {X 0,Y 393.856,Z 772.49,A -85,B 0,C 180,E1 18451.089,E2 18451.089} C_VEL
LIN {X 0,Y 394.428,Z 756.574,A -85,B 0,C 180,E1 18450.484,E2 18450.484} C_VEL
LIN {X 0,Y 395.203,Z 718.668,A -85,B 0,C 180,E1 18449.695,E2 18449.695} C_VEL
LIN {X 0,Y 396.257,Z 657.143,A -85,B 0,C 180,E1 18448.528,E2 18448.528} C_VEL
LIN {X 0,Y 391.578,Z 630.091,A -85,B 0,C 180,E1 18447.657,E2 18447.657} C_VEL
LIN {X 0,Y 394.212,Z 600.99,A -85,B 0,C 180,E1 18443.299,E2 18443.299} C_VEL
LIN {X 0,Y 397.091,Z 573.494,A -85,B 0,C 180,E1 18439.114,E2 18439.114} C_VEL
LIN {X 0,Y 397.05,Z 570.785,A -85,B 0,C 180,E1 18438.671,E2 18438.671} C_VEL
LIN {X 0,Y 392.503,Z 553.654,A -85,B 0,C 180,E1 18435.392,E2 18435.392} C_VEL
LIN {X 0,Y 387.94,Z 538.401,A -85,B 0,C 180,E1 18432.294,E2 18432.294} C_VEL
LIN {X 0,Y 385.573,Z 530.89,A -85,B 0,C 180,E1 18430.639,E2 18430.639} C_VEL
LIN {X 0,Y 385.564,Z 530.724,A -85,B 0,C 180,E1 18426.786,E2 18426.786} C_VEL
LIN {X 0,Y 385.578,Z 530.767,A -85,B 0,C 180,E1 18422.805,E2 18422.805} C_VEL
LIN {X 0,Y 385.583,Z 530.709,A -85,B 0,C 180,E1 18418.841,E2 18418.841} C_VEL
LIN {X 0,Y 385.59,Z 530.766,A -85,B 0,C 180,E1 18414.768,E2 18414.768} C_VEL
LIN {X 0,Y 385.605,Z 530.764,A -85,B 0,C 180,E1 18410.753,E2 18410.753} C_VEL
LIN {X 0,Y 385.587,Z 530.746,A -85,B 0,C 180,E1 18406.774,E2 18406.774} C_VEL
LIN {X 0,Y 385.579,Z 530.757,A -85,B 0,C 180,E1 18402.792,E2 18402.792} C_VEL
LIN {X 0,Y 385.57,Z 530.762,A -85,B 0,C 180,E1 18398.87,E2 18398.87} C_VEL
LIN {X 0,Y 385.559,Z 530.747,A -85,B 0,C 180,E1 18394.968,E2 18394.968} C_VEL
LIN {X 0,Y 385.56,Z 530.766,A -85,B 0,C 180,E1 18391.069,E2 18391.069} C_VEL
LIN {X 0,Y 385.558,Z 530.743,A -85,B 0,C 180,E1 18386.99,E2 18386.99} C_VEL
LIN {X 0,Y 385.563,Z 530.765,A -85,B 0,C 180,E1 18382.892,E2 18382.892} C_VEL
LIN {X 0,Y 385.564,Z 530.745,A -85,B 0,C 180,E1 18378.83,E2 18378.83} C_VEL
LIN {X 0,Y 385.571,Z 530.762,A -85,B 0,C 180,E1 18374.876,E2 18374.876} C_VEL
LIN {X 0,Y 385.586,Z 530.752,A -85,B 0,C 180,E1 18371.063,E2 18371.063} C_VEL
LIN {X 0,Y 385.604,Z 530.741,A -85,B 0,C 180,E1 18367.15,E2 18367.15} C_VEL
LIN {X 0,Y 385.609,Z 530.755,A -85,B 0,C 180,E1 18363.122,E2 18363.122} C_VEL
LIN {X 0,Y 385.618,Z 530.734,A -85,B 0,C 180,E1 18359.109,E2 18359.109} C_VEL
LIN {X 0,Y 385.616,Z 530.758,A -85,B 0,C 180,E1 18355.092,E2 18355.092} C_VEL
LIN {X 0,Y 385.612,Z 530.742,A -85,B 0,C 180,E1 18351.05,E2 18351.05} C_VEL
LIN {X 0,Y 385.601,Z 530.756,A -85,B 0,C 180,E1 18347.115,E2 18347.115} C_VEL
LIN {X 0,Y 385.589,Z 530.758,A -85,B 0,C 180,E1 18343.272,E2 18343.272} C_VEL
LIN {X 0,Y 385.581,Z 530.748,A -85,B 0,C 180,E1 18339.35,E2 18339.35} C_VEL
LIN {X 0,Y 385.585,Z 530.766,A -85,B 0,C 180,E1 18335.324,E2 18335.324} C_VEL
LIN {X 0,Y 385.586,Z 530.766,A -85,B 0,C 180,E1 18331.333,E2 18331.333} C_VEL
LIN {X 0,Y 385.59,Z 530.763,A -85,B 0,C 180,E1 18327.36,E2 18327.36} C_VEL
LIN {X 0,Y 385.596,Z 530.763,A -85,B 0,C 180,E1 18323.388,E2 18323.388} C_VEL
LIN {X 0,Y 385.607,Z 530.766,A -85,B 0,C 180,E1 18319.396,E2 18319.396} C_VEL
LIN {X 0,Y 385.61,Z 530.757,A -85,B 0,C 180,E1 18315.357,E2 18315.357} C_VEL
LIN {X 0,Y 385.66,Z 531.126,A -85,B 0,C 180,E1 18314.268,E2 18314.268} C_VEL
LIN {X 0,Y 393.29,Z 551.718,A -85,B 0,C 180,E1 18310.747,E2 18310.747} C_VEL
LIN {X 0,Y 400.787,Z 573.772,A -85,B 0,C 180,E1 18307.385,E2 18307.385} C_VEL
LIN {X 0,Y 402.551,Z 580.094,A -85,B 0,C 180,E1 18306.502,E2 18306.502} C_VEL
LIN {X 0,Y 398.289,Z 617.541,A -85,B 0,C 180,E1 18302.627,E2 18302.627} C_VEL
LIN {X 0,Y 401.038,Z 644.617,A -85,B 0,C 180,E1 18301.91,E2 18301.91} C_VEL
LIN {X 0,Y 397.834,Z 813.922,A -85,B 0,C 180,E1 18298.876,E2 18298.876} C_VEL
LIN {X 0,Y 396.825,Z 832.508,A -85,B 0,C 180,E1 18298.294,E2 18298.294} C_VEL
LIN {X 0,Y 395.436,Z 850.975,A -85,B 0,C 180,E1 18297.439,E2 18297.439} C_VEL
LIN {X 0,Y 393.837,Z 868.539,A -85,B 0,C 180,E1 18296.339,E2 18296.339} C_VEL
LIN {X 0,Y 392.189,Z 884.786,A -85,B 0,C 180,E1 18295.037,E2 18295.037} C_VEL
LIN {X 0,Y 390.421,Z 900.59,A -85,B 0,C 180,E1 18293.467,E2 18293.467} C_VEL
LIN {X 0,Y 388.791,Z 915.465,A -85,B 0,C 180,E1 18291.656,E2 18291.656} C_VEL
LIN {X 0,Y 387.302,Z 929.299,A -85,B 0,C 180,E1 18289.61,E2 18289.61} C_VEL
LIN {X 0,Y 386.076,Z 941.918,A -85,B 0,C 180,E1 18287.327,E2 18287.327} C_VEL
LIN {X 0,Y 385.266,Z 952.318,A -85,B 0,C 180,E1 18285.042,E2 18285.042} C_VEL
LIN {X 0,Y 384.769,Z 961.341,A -85,B 0,C 180,E1 18282.609,E2 18282.609} C_VEL
LIN {X 0,Y 384.595,Z 968.904,A -85,B 0,C 180,E1 18280.032,E2 18280.032} C_VEL
LIN {X 0,Y 384.639,Z 974.607,A -85,B 0,C 180,E1 18277.469,E2 18277.469} C_VEL
LIN {X 0,Y 384.811,Z 978.584,A -85,B 0,C 180,E1 18274.92,E2 18274.92} C_VEL
LIN {X 0,Y 384.972,Z 980.917,A -85,B 0,C 180,E1 18272.383,E2 18272.383} C_VEL
LIN {X 0,Y 385.036,Z 981.649,A -85,B 0,C 180,E1 18269.853,E2 18269.853} C_VEL
LIN {X 0,Y 384.953,Z 980.76,A -85,B 0,C 180,E1 18267.322,E2 18267.322} C_VEL
LIN {X 0,Y 384.78,Z 978.275,A -85,B 0,C 180,E1 18264.784,E2 18264.784} C_VEL
LIN {X 0,Y 384.607,Z 974.172,A -85,B 0,C 180,E1 18262.233,E2 18262.233} C_VEL
LIN {X 0,Y 384.582,Z 968.378,A -85,B 0,C 180,E1 18259.669,E2 18259.669} C_VEL
LIN {X 0,Y 384.8,Z 960.489,A -85,B 0,C 180,E1 18257.006,E2 18257.006} C_VEL
LIN {X 0,Y 385.386,Z 951.135,A -85,B 0,C 180,E1 18254.504,E2 18254.504} C_VEL
LIN {X 0,Y 386.365,Z 939.909,A -85,B 0,C 180,E1 18252.067,E2 18252.067} C_VEL
LIN {X 0,Y 387.746,Z 927.045,A -85,B 0,C 180,E1 18249.789,E2 18249.789} C_VEL
LIN {X 0,Y 389.392,Z 913.068,A -85,B 0,C 180,E1 18247.748,E2 18247.748} C_VEL
LIN {X 0,Y 391.181,Z 898.28,A -85,B 0,C 180,E1 18245.963,E2 18245.963} C_VEL
LIN {X 0,Y 393.151,Z 882.253,A -85,B 0,C 180,E1 18244.388,E2 18244.388} C_VEL
LIN {X 0,Y 395.013,Z 865.441,A -85,B 0,C 180,E1 18243.063,E2 18243.063} C_VEL
LIN {X 0,Y 396.699,Z 848.437,A -85,B 0,C 180,E1 18242.019,E2 18242.019} C_VEL
LIN {X 0,Y 398.201,Z 830.387,A -85,B 0,C 180,E1 18241.199,E2 18241.199} C_VEL
LIN {X 0,Y 399.28,Z 811.55,A -85,B 0,C 180,E1 18240.621,E2 18240.621} C_VEL
LIN {X 0,Y 402.747,Z 641.845,A -85,B 0,C 180,E1 18237.507,E2 18237.507} C_VEL
LIN {X 0,Y 400.087,Z 617.496,A -85,B 0,C 180,E1 18236.738,E2 18236.738} C_VEL
LIN {X 0,Y 404.862,Z 582.087,A -85,B 0,C 180,E1 18232.91,E2 18232.91} C_VEL
LIN {X 0,Y 399.762,Z 566.191,A -85,B 0,C 180,E1 18230.273,E2 18230.273} C_VEL
LIN {X 0,Y 394.375,Z 551.746,A -85,B 0,C 180,E1 18227.542,E2 18227.542} C_VEL
LIN {X 0,Y 389.012,Z 538.806,A -85,B 0,C 180,E1 18224.769,E2 18224.769} C_VEL
LIN {X 0,Y 385.628,Z 531.036,A -85,B 0,C 180,E1 18222.881,E2 18222.881} C_VEL
LIN {X 0,Y 385.59,Z 530.759,A -85,B 0,C 180,E1 18219.635,E2 18219.635} C_VEL
LIN {X 0,Y 385.596,Z 530.753,A -85,B 0,C 180,E1 18215.692,E2 18215.692} C_VEL
LIN {X 0,Y 385.607,Z 530.75,A -85,B 0,C 180,E1 18211.747,E2 18211.747} C_VEL
LIN {X 0,Y 385.617,Z 530.747,A -85,B 0,C 180,E1 18207.821,E2 18207.821} C_VEL
LIN {X 0,Y 385.606,Z 530.746,A -85,B 0,C 180,E1 18203.697,E2 18203.697} C_VEL
LIN {X 0,Y 385.597,Z 530.748,A -85,B 0,C 180,E1 18199.7,E2 18199.7} C_VEL
LIN {X 0,Y 385.594,Z 530.753,A -85,B 0,C 180,E1 18195.645,E2 18195.645} C_VEL
LIN {X 0,Y 385.576,Z 530.77,A -85,B 0,C 180,E1 18191.669,E2 18191.669} C_VEL
LIN {X 0,Y 385.565,Z 530.766,A -85,B 0,C 180,E1 18187.75,E2 18187.75} C_VEL
LIN {X 0,Y 385.556,Z 530.752,A -85,B 0,C 180,E1 18183.866,E2 18183.866} C_VEL
LIN {X 0,Y 385.554,Z 530.749,A -85,B 0,C 180,E1 18180,E2 18180} C_VEL
LIN {X 0,Y 385.56,Z 530.758,A -85,B 0,C 180,E1 18175.985,E2 18175.985} C_VEL
LIN {X 0,Y 385.569,Z 530.765,A -85,B 0,C 180,E1 18171.95,E2 18171.95} C_VEL
LIN {X 0,Y 385.574,Z 530.768,A -85,B 0,C 180,E1 18167.875,E2 18167.875} C_VEL
LIN {X 0,Y 385.581,Z 530.767,A -85,B 0,C 180,E1 18163.891,E2 18163.891} C_VEL
LIN {X 0,Y 385.594,Z 530.761,A -85,B 0,C 180,E1 18159.984,E2 18159.984} C_VEL
LIN {X 0,Y 385.612,Z 530.753,A -85,B 0,C 180,E1 18156.14,E2 18156.14} C_VEL
LIN {X 0,Y 385.66,Z 531.021,A -85,B 0,C 180,E1 18152.476,E2 18152.476} C_VEL
LIN {X 0,Y 389.741,Z 542.078,A -85,B 0,C 180,E1 18149.472,E2 18149.472} C_VEL
LIN {X 0,Y 393.817,Z 553.868,A -85,B 0,C 180,E1 18146.568,E2 18146.568} C_VEL
LIN {X 0,Y 397.811,Z 567.414,A -85,B 0,C 180,E1 18143.532,E2 18143.532} C_VEL
LIN {X 0,Y 400.007,Z 576.811,A -85,B 0,C 180,E1 18141.599,E2 18141.599} C_VEL
LIN {X 0,Y 396.564,Z 603.452,A -85,B 0,C 180,E1 18137.402,E2 18137.402} C_VEL
LIN {X 0,Y 393.701,Z 629.991,A -85,B 0,C 180,E1 18133.313,E2 18133.313} C_VEL
LIN {X 0,Y 399.122,Z 658.141,A -85,B 0,C 180,E1 18132.205,E2 18132.205} C_VEL
LIN {X 0,Y 399.18,Z 666.111,A -85,B 0,C 180,E1 18132.032,E2 18132.032} C_VEL
LIN {X 0,Y 396.874,Z 756.053,A -85,B 0,C 180,E1 18130.223,E2 18130.223} C_VEL
LIN {X 0,Y 396.217,Z 772.416,A -85,B 0,C 180,E1 18129.611,E2 18129.611} C_VEL
LIN {X 0,Y 395.322,Z 786.472,A -85,B 0,C 180,E1 18128.83,E2 18128.83} C_VEL
LIN {X 0,Y 394.031,Z 801.443,A -85,B 0,C 180,E1 18127.695,E2 18127.695} C_VEL
LIN {X 0,Y 392.607,Z 814.448,A -85,B 0,C 180,E1 18126.392,E2 18126.392} C_VEL
LIN {X 0,Y 391.155,Z 826.423,A -85,B 0,C 180,E1 18124.861,E2 18124.861} C_VEL
LIN {X 0,Y 389.654,Z 837.534,A -85,B 0,C 180,E1 18123.038,E2 18123.038} C_VEL
LIN {X 0,Y 388.376,Z 846.458,A -85,B 0,C 180,E1 18121.157,E2 18121.157} C_VEL
LIN {X 0,Y 387.255,Z 854.198,A -85,B 0,C 180,E1 18119.034,E2 18119.034} C_VEL
LIN {X 0,Y 386.397,Z 860.177,A -85,B 0,C 180,E1 18116.755,E2 18116.755} C_VEL
LIN {X 0,Y 385.842,Z 864.159,A -85,B 0,C 180,E1 18114.491,E2 18114.491} C_VEL
LIN {X 0,Y 385.504,Z 866.445,A -85,B 0,C 180,E1 18112.087,E2 18112.087} C_VEL
LIN {X 0,Y 385.376,Z 866.812,A -85,B 0,C 180,E1 18109.708,E2 18109.708} C_VEL
LIN {X 0,Y 385.442,Z 865.391,A -85,B 0,C 180,E1 18107.327,E2 18107.327} C_VEL
LIN {X 0,Y 385.725,Z 861.9,A -85,B 0,C 180,E1 18104.867,E2 18104.867} C_VEL
LIN {X 0,Y 386.184,Z 857.001,A -85,B 0,C 180,E1 18102.71,E2 18102.71} C_VEL
LIN {X 0,Y 386.899,Z 850.266,A -85,B 0,C 180,E1 18100.57,E2 18100.57} C_VEL
LIN {X 0,Y 387.82,Z 841.971,A -85,B 0,C 180,E1 18098.597,E2 18098.597} C_VEL
LIN {X 0,Y 388.908,Z 832.274,A -85,B 0,C 180,E1 18096.789,E2 18096.789} C_VEL
LIN {X 0,Y 390.16,Z 820.474,A -85,B 0,C 180,E1 18095.07,E2 18095.07} C_VEL
LIN {X 0,Y 390.744,Z 814.515,A -85,B 0,C 180,E1 18094.346,E2 18094.346} C_VEL
LIN {X 0,Y 390.362,Z 808.487,A -85,B 0,C 180,E1 18093.643,E2 18093.643} C_VEL
LIN {X 0,Y 386.719,Z 795.458,A -85,B 0,C 180,E1 18092.185,E2 18092.185} C_VEL
LIN {X 0,Y 385.646,Z 787.781,A -85,B 0,C 180,E1 18091.526,E2 18091.526} C_VEL
LIN {X 0,Y 385.662,Z 785.763,A -85,B 0,C 180,E1 18091.386,E2 18091.386} C_VEL
LIN {X 0,Y 386.501,Z 770.859,A -85,B 0,C 180,E1 18090.568,E2 18090.568} C_VEL
LIN {X 0,Y 387.075,Z 754.678,A -85,B 0,C 180,E1 18089.98,E2 18089.98} C_VEL
LIN {X 0,Y 388.949,Z 658.35,A -85,B 0,C 180,E1 18088.074,E2 18088.074} C_VEL
LIN {X 0,Y 384.108,Z 630.326,A -85,B 0,C 180,E1 18087.164,E2 18087.164} C_VEL
LIN {X 0,Y 384.585,Z 624.081,A -85,B 0,C 180,E1 18086.272,E2 18086.272} C_VEL
LIN {X 0,Y 387.373,Z 596.123,A -85,B 0,C 180,E1 18081.987,E2 18081.987} C_VEL
LIN {X 0,Y 389.732,Z 573.867,A -85,B 0,C 180,E1 18078.53,E2 18078.53} C_VEL
LIN {X 0,Y 385.09,Z 556.237,A -85,B 0,C 180,E1 18075.105,E2 18075.105} C_VEL
LIN {X 0,Y 380.195,Z 539.844,A -85,B 0,C 180,E1 18071.693,E2 18071.693} C_VEL
LIN {X 0,Y 377.64,Z 531.889,A -85,B 0,C 180,E1 18069.908,E2 18069.908} C_VEL
LIN {X 0,Y 377.608,Z 531.713,A -85,B 0,C 180,E1 18065.935,E2 18065.935} C_VEL
LIN {X 0,Y 377.607,Z 531.744,A -85,B 0,C 180,E1 18062.052,E2 18062.052} C_VEL
LIN {X 0,Y 377.601,Z 531.715,A -85,B 0,C 180,E1 18057.924,E2 18057.924} C_VEL
LIN {X 0,Y 377.608,Z 531.751,A -85,B 0,C 180,E1 18053.811,E2 18053.811} C_VEL
LIN {X 0,Y 377.61,Z 531.759,A -85,B 0,C 180,E1 18049.693,E2 18049.693} C_VEL
LIN {X 0,Y 377.614,Z 531.755,A -85,B 0,C 180,E1 18045.637,E2 18045.637} C_VEL
LIN {X 0,Y 377.615,Z 531.734,A -85,B 0,C 180,E1 18041.653,E2 18041.653} C_VEL
LIN {X 0,Y 377.624,Z 531.758,A -85,B 0,C 180,E1 18037.66,E2 18037.66} C_VEL
LIN {X 0,Y 377.635,Z 531.727,A -85,B 0,C 180,E1 18033.764,E2 18033.764} C_VEL
LIN {X 0,Y 377.656,Z 531.754,A -85,B 0,C 180,E1 18029.851,E2 18029.851} C_VEL
LIN {X 0,Y 377.659,Z 531.72,A -85,B 0,C 180,E1 18025.828,E2 18025.828} C_VEL
LIN {X 0,Y 377.669,Z 531.753,A -85,B 0,C 180,E1 18021.689,E2 18021.689} C_VEL
LIN {X 0,Y 377.663,Z 531.716,A -85,B 0,C 180,E1 18017.567,E2 18017.567} C_VEL
LIN {X 0,Y 377.673,Z 531.754,A -85,B 0,C 180,E1 18013.473,E2 18013.473} C_VEL
LIN {X 0,Y 377.669,Z 531.714,A -85,B 0,C 180,E1 18009.448,E2 18009.448} C_VEL
LIN {X 0,Y 377.669,Z 531.748,A -85,B 0,C 180,E1 18005.469,E2 18005.469} C_VEL
LIN {X 0,Y 377.668,Z 531.719,A -85,B 0,C 180,E1 18001.366,E2 18001.366} C_VEL
LIN {X 0,Y 377.66,Z 531.748,A -85,B 0,C 180,E1 17997.421,E2 17997.421} C_VEL
LIN {X 0,Y 377.649,Z 531.73,A -85,B 0,C 180,E1 17993.463,E2 17993.463} C_VEL
LIN {X 0,Y 377.647,Z 531.752,A -85,B 0,C 180,E1 17989.474,E2 17989.474} C_VEL
LIN {X 0,Y 377.641,Z 531.731,A -85,B 0,C 180,E1 17985.432,E2 17985.432} C_VEL
LIN {X 0,Y 377.646,Z 531.756,A -85,B 0,C 180,E1 17981.405,E2 17981.405} C_VEL
LIN {X 0,Y 377.644,Z 531.747,A -85,B 0,C 180,E1 17977.424,E2 17977.424} C_VEL
LIN {X 0,Y 377.646,Z 531.735,A -85,B 0,C 180,E1 17973.42,E2 17973.42} C_VEL
LIN {X 0,Y 377.648,Z 531.745,A -85,B 0,C 180,E1 17969.364,E2 17969.364} C_VEL
LIN {X 0,Y 377.649,Z 531.747,A -85,B 0,C 180,E1 17965.304,E2 17965.304} C_VEL
LIN {X 0,Y 377.658,Z 531.744,A -85,B 0,C 180,E1 17961.332,E2 17961.332} C_VEL
LIN {X 0,Y 377.665,Z 531.746,A -85,B 0,C 180,E1 17957.332,E2 17957.332} C_VEL
LIN {X 0,Y 377.689,Z 531.948,A -85,B 0,C 180,E1 17955.13,E2 17955.13} C_VEL
LIN {X 0,Y 383.941,Z 548.858,A -85,B 0,C 180,E1 17952.081,E2 17952.081} C_VEL
LIN {X 0,Y 390.527,Z 567.628,A -85,B 0,C 180,E1 17949.036,E2 17949.036} C_VEL
LIN {X 0,Y 395.176,Z 582.427,A -85,B 0,C 180,E1 17946.843,E2 17946.843} C_VEL
LIN {X 0,Y 390.963,Z 617.515,A -85,B 0,C 180,E1 17943.136,E2 17943.136} C_VEL
LIN {X 0,Y 393.734,Z 645.487,A -85,B 0,C 180,E1 17942.371,E2 17942.371} C_VEL
LIN {X 0,Y 390.392,Z 813.339,A -85,B 0,C 180,E1 17939.31,E2 17939.31} C_VEL
LIN {X 0,Y 389.355,Z 831.864,A -85,B 0,C 180,E1 17938.72,E2 17938.72} C_VEL
LIN {X 0,Y 387.936,Z 850.019,A -85,B 0,C 180,E1 17937.867,E2 17937.867} C_VEL
LIN {X 0,Y 386.257,Z 867.753,A -85,B 0,C 180,E1 17936.74,E2 17936.74} C_VEL
LIN {X 0,Y 384.534,Z 884.121,A -85,B 0,C 180,E1 17935.406,E2 17935.406} C_VEL
LIN {X 0,Y 382.691,Z 899.924,A -85,B 0,C 180,E1 17933.807,E2 17933.807} C_VEL
LIN {X 0,Y 380.986,Z 914.781,A -85,B 0,C 180,E1 17931.961,E2 17931.961} C_VEL
LIN {X 0,Y 379.435,Z 928.547,A -85,B 0,C 180,E1 17929.873,E2 17929.873} C_VEL
LIN {X 0,Y 378.157,Z 941.109,A -85,B 0,C 180,E1 17927.543,E2 17927.543} C_VEL
LIN {X 0,Y 377.314,Z 951.461,A -85,B 0,C 180,E1 17925.21,E2 17925.21} C_VEL
LIN {X 0,Y 376.8,Z 960.435,A -85,B 0,C 180,E1 17922.724,E2 17922.724} C_VEL
LIN {X 0,Y 376.633,Z 967.95,A -85,B 0,C 180,E1 17920.092,E2 17920.092} C_VEL
LIN {X 0,Y 376.693,Z 973.601,A -85,B 0,C 180,E1 17917.474,E2 17917.474} C_VEL
LIN {X 0,Y 376.889,Z 977.522,A -85,B 0,C 180,E1 17914.871,E2 17914.871} C_VEL
LIN {X 0,Y 377.065,Z 979.789,A -85,B 0,C 180,E1 17912.281,E2 17912.281} C_VEL
LIN {X 0,Y 377.121,Z 980.446,A -85,B 0,C 180,E1 17909.698,E2 17909.698} C_VEL
LIN {X 0,Y 377.018,Z 979.498,A -85,B 0,C 180,E1 17907.114,E2 17907.114} C_VEL
LIN {X 0,Y 376.814,Z 976.926,A -85,B 0,C 180,E1 17904.521,E2 17904.521} C_VEL
LIN {X 0,Y 376.625,Z 972.443,A -85,B 0,C 180,E1 17901.76,E2 17901.76} C_VEL
LIN {X 0,Y 376.624,Z 966.024,A -85,B 0,C 180,E1 17898.983,E2 17898.983} C_VEL
LIN {X 0,Y 376.919,Z 958.042,A -85,B 0,C 180,E1 17896.347,E2 17896.347} C_VEL
LIN {X 0,Y 377.59,Z 948.635,A -85,B 0,C 180,E1 17893.86,E2 17893.86} C_VEL
LIN {X 0,Y 378.709,Z 937.076,A -85,B 0,C 180,E1 17891.373,E2 17891.373} C_VEL
LIN {X 0,Y 380.262,Z 923.915,A -85,B 0,C 180,E1 17889.051,E2 17889.051} C_VEL
LIN {X 0,Y 382.081,Z 909.577,A -85,B 0,C 180,E1 17886.973,E2 17886.973} C_VEL
LIN {X 0,Y 384,Z 894.834,A -85,B 0,C 180,E1 17885.22,E2 17885.22} C_VEL
LIN {X 0,Y 386.086,Z 878.531,A -85,B 0,C 180,E1 17883.643,E2 17883.643} C_VEL
LIN {X 0,Y 387.995,Z 862.002,A -85,B 0,C 180,E1 17882.368,E2 17882.368} C_VEL
LIN {X 0,Y 389.8,Z 844.164,A -85,B 0,C 180,E1 17881.312,E2 17881.312} C_VEL
LIN {X 0,Y 391.294,Z 825.996,A -85,B 0,C 180,E1 17880.535,E2 17880.535} C_VEL
LIN {X 0,Y 392.261,Z 807.387,A -85,B 0,C 180,E1 17880.011,E2 17880.011} C_VEL
LIN {X 0,Y 395.824,Z 642.703,A -85,B 0,C 180,E1 17876.938,E2 17876.938} C_VEL
LIN {X 0,Y 393.112,Z 617.668,A -85,B 0,C 180,E1 17876.123,E2 17876.123} C_VEL
LIN {X 0,Y 397.844,Z 585.213,A -85,B 0,C 180,E1 17872.547,E2 17872.547} C_VEL
LIN {X 0,Y 392.979,Z 569.885,A -85,B 0,C 180,E1 17869.938,E2 17869.938} C_VEL
LIN {X 0,Y 387.543,Z 555.181,A -85,B 0,C 180,E1 17867.076,E2 17867.076} C_VEL
LIN {X 0,Y 382.603,Z 543.298,A -85,B 0,C 180,E1 17864.456,E2 17864.456} C_VEL
LIN {X 0,Y 378.686,Z 534.749,A -85,B 0,C 180,E1 17862.321,E2 17862.321} C_VEL
LIN {X 0,Y 377.671,Z 531.913,A -85,B 0,C 180,E1 17861.543,E2 17861.543} C_VEL
LIN {X 0,Y 377.658,Z 531.751,A -85,B 0,C 180,E1 17857.673,E2 17857.673} C_VEL
LIN {X 0,Y 377.656,Z 531.756,A -85,B 0,C 180,E1 17853.596,E2 17853.596} C_VEL
LIN {X 0,Y 377.668,Z 531.753,A -85,B 0,C 180,E1 17849.674,E2 17849.674} C_VEL
LIN {X 0,Y 377.666,Z 531.756,A -85,B 0,C 180,E1 17845.733,E2 17845.733} C_VEL
LIN {X 0,Y 377.671,Z 531.755,A -85,B 0,C 180,E1 17841.592,E2 17841.592} C_VEL
LIN {X 0,Y 377.655,Z 531.751,A -85,B 0,C 180,E1 17837.408,E2 17837.408} C_VEL
LIN {X 0,Y 377.652,Z 531.739,A -85,B 0,C 180,E1 17833.317,E2 17833.317} C_VEL
LIN {X 0,Y 377.65,Z 531.734,A -85,B 0,C 180,E1 17829.294,E2 17829.294} C_VEL
LIN {X 0,Y 377.652,Z 531.736,A -85,B 0,C 180,E1 17825.317,E2 17825.317} C_VEL
LIN {X 0,Y 377.66,Z 531.745,A -85,B 0,C 180,E1 17821.213,E2 17821.213} C_VEL
LIN {X 0,Y 377.66,Z 531.755,A -85,B 0,C 180,E1 17817.116,E2 17817.116} C_VEL
LIN {X 0,Y 377.672,Z 531.753,A -85,B 0,C 180,E1 17813.005,E2 17813.005} C_VEL
LIN {X 0,Y 377.671,Z 531.751,A -85,B 0,C 180,E1 17808.856,E2 17808.856} C_VEL
LIN {X 0,Y 377.678,Z 531.75,A -85,B 0,C 180,E1 17804.805,E2 17804.805} C_VEL
LIN {X 0,Y 377.68,Z 531.755,A -85,B 0,C 180,E1 17800.675,E2 17800.675} C_VEL
LIN {X 0,Y 377.683,Z 531.745,A -85,B 0,C 180,E1 17796.602,E2 17796.602} C_VEL
LIN {X 0,Y 377.695,Z 532.03,A -85,B 0,C 180,E1 17793.709,E2 17793.709} C_VEL
LIN {X 0,Y 381.948,Z 543.136,A -85,B 0,C 180,E1 17790.518,E2 17790.518} C_VEL
LIN {X 0,Y 386.169,Z 555.168,A -85,B 0,C 180,E1 17787.415,E2 17787.415} C_VEL
LIN {X 0,Y 390.133,Z 568.425,A -85,B 0,C 180,E1 17784.324,E2 17784.324} C_VEL
LIN {X 0,Y 392.825,Z 579.706,A -85,B 0,C 180,E1 17781.923,E2 17781.923} C_VEL
LIN {X 0,Y 389.229,Z 606.106,A -85,B 0,C 180,E1 17777.698,E2 17777.698} C_VEL
LIN {X 0,Y 386.527,Z 629.524,A -85,B 0,C 180,E1 17774.017,E2 17774.017} C_VEL
LIN {X 0,Y 387.588,Z 635.188,A -85,B 0,C 180,E1 17773.729,E2 17773.729} C_VEL
LIN {X 0,Y 392.437,Z 661.167,A -85,B 0,C 180,E1 17772.721,E2 17772.721} C_VEL
LIN {X 0,Y 389.855,Z 756.325,A -85,B 0,C 180,E1 17770.782,E2 17770.782} C_VEL
LIN {X 0,Y 389.181,Z 772.361,A -85,B 0,C 180,E1 17770.181,E2 17770.181} C_VEL
LIN {X 0,Y 388.21,Z 786.968,A -85,B 0,C 180,E1 17769.367,E2 17769.367} C_VEL
LIN {X 0,Y 386.829,Z 802.042,A -85,B 0,C 180,E1 17768.208,E2 17768.208} C_VEL
LIN {X 0,Y 385.35,Z 814.851,A -85,B 0,C 180,E1 17766.912,E2 17766.912} C_VEL
LIN {X 0,Y 383.77,Z 827.096,A -85,B 0,C 180,E1 17765.332,E2 17765.332} C_VEL
LIN {X 0,Y 382.181,Z 838.142,A -85,B 0,C 180,E1 17763.5,E2 17763.5} C_VEL
LIN {X 0,Y 380.86,Z 846.852,A -85,B 0,C 180,E1 17761.667,E2 17761.667} C_VEL
LIN {X 0,Y 379.616,Z 854.742,A -85,B 0,C 180,E1 17759.502,E2 17759.502} C_VEL
LIN {X 0,Y 378.718,Z 860.552,A -85,B 0,C 180,E1 17757.342,E2 17757.342} C_VEL
LIN {X 0,Y 378.066,Z 864.836,A -85,B 0,C 180,E1 17755.029,E2 17755.029} C_VEL
LIN {X 0,Y 377.67,Z 867.284,A -85,B 0,C 180,E1 17752.734,E2 17752.734} C_VEL
LIN {X 0,Y 377.483,Z 868.093,A -85,B 0,C 180,E1 17750.299,E2 17750.299} C_VEL
LIN {X 0,Y 377.492,Z 867.06,A -85,B 0,C 180,E1 17747.89,E2 17747.89} C_VEL
LIN {X 0,Y 377.717,Z 864.272,A -85,B 0,C 180,E1 17745.504,E2 17745.504} C_VEL
LIN {X 0,Y 378.166,Z 859.557,A -85,B 0,C 180,E1 17743.14,E2 17743.14} C_VEL
LIN {X 0,Y 378.842,Z 853.278,A -85,B 0,C 180,E1 17740.945,E2 17740.945} C_VEL
LIN {X 0,Y 379.823,Z 844.951,A -85,B 0,C 180,E1 17738.78,E2 17738.78} C_VEL
LIN {X 0,Y 381.01,Z 834.833,A -85,B 0,C 180,E1 17736.779,E2 17736.779} C_VEL
LIN {X 0,Y 382.234,Z 824.011,A -85,B 0,C 180,E1 17735.1,E2 17735.1} C_VEL
LIN {X 0,Y 383.509,Z 811.661,A -85,B 0,C 180,E1 17733.585,E2 17733.585} C_VEL
LIN {X 0,Y 384.703,Z 798.587,A -85,B 0,C 180,E1 17732.338,E2 17732.338} C_VEL
LIN {X 0,Y 385.662,Z 785.763,A -85,B 0,C 180,E1 17731.386,E2 17731.386} C_VEL
LIN {X 0,Y 385.212,Z 778.728,A -85,B 0,C 180,E1 17730.898,E2 17730.898} C_VEL
LIN {X 0,Y 381.744,Z 765.856,A -85,B 0,C 180,E1 17730.031,E2 17730.031} C_VEL
LIN {X 0,Y 379.969,Z 757.572,A -85,B 0,C 180,E1 17729.621,E2 17729.621} C_VEL
LIN {X 0,Y 379.715,Z 753.245,A -85,B 0,C 180,E1 17729.482,E2 17729.482} C_VEL
LIN {X 0,Y 381.629,Z 659.333,A -85,B 0,C 180,E1 17727.596,E2 17727.596} C_VEL
LIN {X 0,Y 376.614,Z 629.784,A -85,B 0,C 180,E1 17726.598,E2 17726.598} C_VEL
LIN {X 0,Y 379.427,Z 601.792,A -85,B 0,C 180,E1 17722.275,E2 17722.275} C_VEL
LIN {X 0,Y 382.319,Z 576.544,A -85,B 0,C 180,E1 17718.305,E2 17718.305} C_VEL
LIN {X 0,Y 377.896,Z 559.603,A -85,B 0,C 180,E1 17714.96,E2 17714.96} C_VEL
LIN {X 0,Y 373.13,Z 543.503,A -85,B 0,C 180,E1 17711.551,E2 17711.551} C_VEL
LIN {X 0,Y 369.722,Z 532.83,A -85,B 0,C 180,E1 17709.085,E2 17709.085} C_VEL
LIN {X 0,Y 369.706,Z 532.706,A -85,B 0,C 180,E1 17705.046,E2 17705.046} C_VEL
LIN {X 0,Y 369.712,Z 532.697,A -85,B 0,C 180,E1 17701.048,E2 17701.048} C_VEL
LIN {X 0,Y 369.71,Z 532.724,A -85,B 0,C 180,E1 17696.888,E2 17696.888} C_VEL
LIN {X 0,Y 369.711,Z 532.726,A -85,B 0,C 180,E1 17692.716,E2 17692.716} C_VEL
LIN {X 0,Y 369.719,Z 532.73,A -85,B 0,C 180,E1 17688.712,E2 17688.712} C_VEL
LIN {X 0,Y 369.714,Z 532.745,A -85,B 0,C 180,E1 17684.665,E2 17684.665} C_VEL
LIN {X 0,Y 369.722,Z 532.717,A -85,B 0,C 180,E1 17680.47,E2 17680.47} C_VEL
LIN {X 0,Y 369.718,Z 532.735,A -85,B 0,C 180,E1 17676.318,E2 17676.318} C_VEL
LIN {X 0,Y 369.723,Z 532.727,A -85,B 0,C 180,E1 17672.176,E2 17672.176} C_VEL
LIN {X 0,Y 369.728,Z 532.725,A -85,B 0,C 180,E1 17668.07,E2 17668.07} C_VEL
LIN {X 0,Y 369.728,Z 532.726,A -85,B 0,C 180,E1 17663.932,E2 17663.932} C_VEL
LIN {X 0,Y 369.723,Z 532.728,A -85,B 0,C 180,E1 17659.923,E2 17659.923} C_VEL
LIN {X 0,Y 369.733,Z 532.719,A -85,B 0,C 180,E1 17655.69,E2 17655.69} C_VEL
LIN {X 0,Y 369.724,Z 532.734,A -85,B 0,C 180,E1 17651.703,E2 17651.703} C_VEL
LIN {X 0,Y 369.723,Z 532.708,A -85,B 0,C 180,E1 17647.615,E2 17647.615} C_VEL
LIN {X 0,Y 369.721,Z 532.739,A -85,B 0,C 180,E1 17643.566,E2 17643.566} C_VEL
LIN {X 0,Y 369.712,Z 532.707,A -85,B 0,C 180,E1 17639.535,E2 17639.535} C_VEL
LIN {X 0,Y 369.713,Z 532.745,A -85,B 0,C 180,E1 17635.502,E2 17635.502} C_VEL
LIN {X 0,Y 369.702,Z 532.715,A -85,B 0,C 180,E1 17631.603,E2 17631.603} C_VEL
LIN {X 0,Y 369.706,Z 532.742,A -85,B 0,C 180,E1 17627.505,E2 17627.505} C_VEL
LIN {X 0,Y 369.704,Z 532.735,A -85,B 0,C 180,E1 17623.503,E2 17623.503} C_VEL
LIN {X 0,Y 369.704,Z 532.725,A -85,B 0,C 180,E1 17619.416,E2 17619.416} C_VEL
LIN {X 0,Y 369.708,Z 532.744,A -85,B 0,C 180,E1 17615.319,E2 17615.319} C_VEL
LIN {X 0,Y 369.71,Z 532.744,A -85,B 0,C 180,E1 17611.187,E2 17611.187} C_VEL
LIN {X 0,Y 369.712,Z 532.742,A -85,B 0,C 180,E1 17607.072,E2 17607.072} C_VEL
LIN {X 0,Y 369.713,Z 532.745,A -85,B 0,C 180,E1 17602.909,E2 17602.909} C_VEL
LIN {X 0,Y 369.716,Z 532.74,A -85,B 0,C 180,E1 17598.746,E2 17598.746} C_VEL
LIN {X 0,Y 369.79,Z 533.047,A -85,B 0,C 180,E1 17595.928,E2 17595.928} C_VEL
LIN {X 0,Y 376.78,Z 551.775,A -85,B 0,C 180,E1 17592.462,E2 17592.462} C_VEL
LIN {X 0,Y 383.501,Z 571.16,A -85,B 0,C 180,E1 17589.256,E2 17589.256} C_VEL
LIN {X 0,Y 387.78,Z 584.85,A -85,B 0,C 180,E1 17587.181,E2 17587.181} C_VEL
LIN {X 0,Y 383.645,Z 617.783,A -85,B 0,C 180,E1 17583.638,E2 17583.638} C_VEL
LIN {X 0,Y 386.451,Z 646.395,A -85,B 0,C 180,E1 17582.849,E2 17582.849} C_VEL
LIN {X 0,Y 382.975,Z 812.706,A -85,B 0,C 180,E1 17579.763,E2 17579.763} C_VEL
LIN {X 0,Y 381.909,Z 831.221,A -85,B 0,C 180,E1 17579.162,E2 17579.162} C_VEL
LIN {X 0,Y 380.452,Z 849.097,A -85,B 0,C 180,E1 17578.309,E2 17578.309} C_VEL
LIN {X 0,Y 378.696,Z 866.944,A -85,B 0,C 180,E1 17577.156,E2 17577.156} C_VEL
LIN {X 0,Y 376.892,Z 883.385,A -85,B 0,C 180,E1 17575.79,E2 17575.79} C_VEL
LIN {X 0,Y 374.97,Z 899.154,A -85,B 0,C 180,E1 17574.161,E2 17574.161} C_VEL
LIN {X 0,Y 373.193,Z 913.989,A -85,B 0,C 180,E1 17572.278,E2 17572.278} C_VEL
LIN {X 0,Y 371.576,Z 927.741,A -85,B 0,C 180,E1 17570.147,E2 17570.147} C_VEL
LIN {X 0,Y 370.241,Z 940.292,A -85,B 0,C 180,E1 17567.768,E2 17567.768} C_VEL
LIN {X 0,Y 369.362,Z 950.603,A -85,B 0,C 180,E1 17565.384,E2 17565.384} C_VEL
LIN {X 0,Y 368.833,Z 959.529,A -85,B 0,C 180,E1 17562.844,E2 17562.844} C_VEL
LIN {X 0,Y 368.669,Z 967.11,A -85,B 0,C 180,E1 17560.107,E2 17560.107} C_VEL
LIN {X 0,Y 368.759,Z 972.867,A -85,B 0,C 180,E1 17557.323,E2 17557.323} C_VEL
LIN {X 0,Y 368.98,Z 976.629,A -85,B 0,C 180,E1 17554.664,E2 17554.664} C_VEL
LIN {X 0,Y 369.17,Z 978.744,A -85,B 0,C 180,E1 17551.992,E2 17551.992} C_VEL
LIN {X 0,Y 369.208,Z 979.213,A -85,B 0,C 180,E1 17549.381,E2 17549.381} C_VEL
LIN {X 0,Y 369.073,Z 978.085,A -85,B 0,C 180,E1 17546.741,E2 17546.741} C_VEL
LIN {X 0,Y 368.84,Z 975.349,A -85,B 0,C 180,E1 17544.09,E2 17544.09} C_VEL
LIN {X 0,Y 368.647,Z 970.965,A -85,B 0,C 180,E1 17541.424,E2 17541.424} C_VEL
LIN {X 0,Y 368.651,Z 964.846,A -85,B 0,C 180,E1 17538.742,E2 17538.742} C_VEL
LIN {X 0,Y 368.999,Z 956.498,A -85,B 0,C 180,E1 17535.943,E2 17535.943} C_VEL
LIN {X 0,Y 369.766,Z 946.796,A -85,B 0,C 180,E1 17533.347,E2 17533.347} C_VEL
LIN {X 0,Y 371.012,Z 935.115,A -85,B 0,C 180,E1 17530.809,E2 17530.809} C_VEL
LIN {X 0,Y 372.579,Z 922.745,A -85,B 0,C 180,E1 17528.598,E2 17528.598} C_VEL
LIN {X 0,Y 374.433,Z 908.956,A -85,B 0,C 180,E1 17526.559,E2 17526.559} C_VEL
LIN {X 0,Y 376.47,Z 894.293,A -85,B 0,C 180,E1 17524.773,E2 17524.773} C_VEL
LIN {X 0,Y 378.606,Z 878.465,A -85,B 0,C 180,E1 17523.205,E2 17523.205} C_VEL
LIN {X 0,Y 380.662,Z 861.693,A -85,B 0,C 180,E1 17521.874,E2 17521.874} C_VEL
LIN {X 0,Y 382.564,Z 844.137,A -85,B 0,C 180,E1 17520.801,E2 17520.801} C_VEL
LIN {X 0,Y 384.166,Z 825.752,A -85,B 0,C 180,E1 17519.992,E2 17519.992} C_VEL
LIN {X 0,Y 385.195,Z 807.228,A -85,B 0,C 180,E1 17519.453,E2 17519.453} C_VEL
LIN {X 0,Y 388.955,Z 643.575,A -85,B 0,C 180,E1 17516.346,E2 17516.346} C_VEL
LIN {X 0,Y 386.184,Z 617.876,A -85,B 0,C 180,E1 17515.486,E2 17515.486} C_VEL
LIN {X 0,Y 390.757,Z 588.021,A -85,B 0,C 180,E1 17512.119,E2 17512.119} C_VEL
LIN {X 0,Y 385.946,Z 572.807,A -85,B 0,C 180,E1 17509.446,E2 17509.446} C_VEL
LIN {X 0,Y 380.834,Z 558.879,A -85,B 0,C 180,E1 17506.656,E2 17506.656} C_VEL
LIN {X 0,Y 375.71,Z 546.671,A -85,B 0,C 180,E1 17503.854,E2 17503.854} C_VEL
LIN {X 0,Y 371.31,Z 536.665,A -85,B 0,C 180,E1 17501.279,E2 17501.279} C_VEL
LIN {X 0,Y 369.781,Z 532.967,A -85,B 0,C 180,E1 17500.215,E2 17500.215} C_VEL
LIN {X 0,Y 369.724,Z 532.733,A -85,B 0,C 180,E1 17496.313,E2 17496.313} C_VEL
LIN {X 0,Y 369.711,Z 532.73,A -85,B 0,C 180,E1 17492.376,E2 17492.376} C_VEL
LIN {X 0,Y 369.699,Z 532.729,A -85,B 0,C 180,E1 17488.424,E2 17488.424} C_VEL
LIN {X 0,Y 369.687,Z 532.732,A -85,B 0,C 180,E1 17484.444,E2 17484.444} C_VEL
LIN {X 0,Y 369.679,Z 532.741,A -85,B 0,C 180,E1 17480.585,E2 17480.585} C_VEL
LIN {X 0,Y 369.675,Z 532.749,A -85,B 0,C 180,E1 17476.498,E2 17476.498} C_VEL
LIN {X 0,Y 369.672,Z 532.749,A -85,B 0,C 180,E1 17472.337,E2 17472.337} C_VEL
LIN {X 0,Y 369.67,Z 532.739,A -85,B 0,C 180,E1 17468.186,E2 17468.186} C_VEL
LIN {X 0,Y 369.675,Z 532.727,A -85,B 0,C 180,E1 17464.032,E2 17464.032} C_VEL
LIN {X 0,Y 369.677,Z 532.725,A -85,B 0,C 180,E1 17460,E2 17460} C_VEL
LIN {X 0,Y 369.683,Z 532.733,A -85,B 0,C 180,E1 17455.967,E2 17455.967} C_VEL
LIN {X 0,Y 369.69,Z 532.738,A -85,B 0,C 180,E1 17451.793,E2 17451.793} C_VEL
LIN {X 0,Y 369.696,Z 532.74,A -85,B 0,C 180,E1 17447.663,E2 17447.663} C_VEL
LIN {X 0,Y 369.7,Z 532.737,A -85,B 0,C 180,E1 17443.502,E2 17443.502} C_VEL
LIN {X 0,Y 369.705,Z 532.733,A -85,B 0,C 180,E1 17439.415,E2 17439.415} C_VEL
LIN {X 0,Y 369.714,Z 532.782,A -85,B 0,C 180,E1 17435.309,E2 17435.309} C_VEL
LIN {X 0,Y 369.866,Z 533.55,A -85,B 0,C 180,E1 17434.886,E2 17434.886} C_VEL
LIN {X 0,Y 373.996,Z 543.777,A -85,B 0,C 180,E1 17431.757,E2 17431.757} C_VEL
LIN {X 0,Y 378.323,Z 555.97,A -85,B 0,C 180,E1 17428.446,E2 17428.446} C_VEL
LIN {X 0,Y 382.457,Z 569.443,A -85,B 0,C 180,E1 17425.164,E2 17425.164} C_VEL
LIN {X 0,Y 385.7,Z 582.536,A -85,B 0,C 180,E1 17422.281,E2 17422.281} C_VEL
LIN {X 0,Y 381.932,Z 608.71,A -85,B 0,C 180,E1 17418.021,E2 17418.021} C_VEL
LIN {X 0,Y 379.4,Z 629.452,A -85,B 0,C 180,E1 17414.712,E2 17414.712} C_VEL
LIN {X 0,Y 380.589,Z 635.62,A -85,B 0,C 180,E1 17414.391,E2 17414.391} C_VEL
LIN {X 0,Y 385.579,Z 662.215,A -85,B 0,C 180,E1 17413.318,E2 17413.318} C_VEL
LIN {X 0,Y 382.866,Z 757.038,A -85,B 0,C 180,E1 17411.35,E2 17411.35} C_VEL
LIN {X 0,Y 382.153,Z 773.068,A -85,B 0,C 180,E1 17410.739,E2 17410.739} C_VEL
LIN {X 0,Y 381.105,Z 787.943,A -85,B 0,C 180,E1 17409.895,E2 17409.895} C_VEL
LIN {X 0,Y 379.642,Z 803.034,A -85,B 0,C 180,E1 17408.713,E2 17408.713} C_VEL
LIN {X 0,Y 378.141,Z 815.356,A -85,B 0,C 180,E1 17407.45,E2 17407.45} C_VEL
LIN {X 0,Y 376.458,Z 827.629,A -85,B 0,C 180,E1 17405.852,E2 17405.852} C_VEL
LIN {X 0,Y 374.817,Z 838.36,A -85,B 0,C 180,E1 17404.064,E2 17404.064} C_VEL
LIN {X 0,Y 373.378,Z 847.241,A -85,B 0,C 180,E1 17402.196,E2 17402.196} C_VEL
LIN {X 0,Y 372.055,Z 855.01,A -85,B 0,C 180,E1 17400.077,E2 17400.077} C_VEL
LIN {X 0,Y 371.009,Z 861.288,A -85,B 0,C 180,E1 17397.785,E2 17397.785} C_VEL
LIN {X 0,Y 370.265,Z 865.702,A -85,B 0,C 180,E1 17395.423,E2 17395.423} C_VEL
LIN {X 0,Y 369.816,Z 868.336,A -85,B 0,C 180,E1 17393.077,E2 17393.077} C_VEL
LIN {X 0,Y 369.581,Z 869.267,A -85,B 0,C 180,E1 17390.587,E2 17390.587} C_VEL
LIN {X 0,Y 369.568,Z 868.423,A -85,B 0,C 180,E1 17388.124,E2 17388.124} C_VEL
LIN {X 0,Y 369.777,Z 865.788,A -85,B 0,C 180,E1 17385.684,E2 17385.684} C_VEL
LIN {X 0,Y 370.187,Z 861.641,A -85,B 0,C 180,E1 17383.428,E2 17383.428} C_VEL
LIN {X 0,Y 370.909,Z 855.256,A -85,B 0,C 180,E1 17381.031,E2 17381.031} C_VEL
LIN {X 0,Y 371.896,Z 847.124,A -85,B 0,C 180,E1 17378.812,E2 17378.812} C_VEL
LIN {X 0,Y 373.01,Z 838.21,A -85,B 0,C 180,E1 17376.926,E2 17376.926} C_VEL
LIN {X 0,Y 374.39,Z 826.73,A -85,B 0,C 180,E1 17375.026,E2 17375.026} C_VEL
LIN {X 0,Y 375.663,Z 815.043,A -85,B 0,C 180,E1 17373.507,E2 17373.507} C_VEL
LIN {X 0,Y 377.009,Z 801.516,A -85,B 0,C 180,E1 17372.126,E2 17372.126} C_VEL
LIN {X 0,Y 378.197,Z 786.46,A -85,B 0,C 180,E1 17370.967,E2 17370.967} C_VEL
LIN {X 0,Y 379.074,Z 771.557,A -85,B 0,C 180,E1 17370.135,E2 17370.135} C_VEL
LIN {X 0,Y 379.679,Z 755.247,A -85,B 0,C 180,E1 17369.531,E2 17369.531} C_VEL
LIN {X 0,Y 379.715,Z 753.245,A -85,B 0,C 180,E1 17369.482,E2 17369.482} C_VEL
LIN {X 0,Y 378.927,Z 745.674,A -85,B 0,C 180,E1 17369.246,E2 17369.246} C_VEL
LIN {X 0,Y 373.684,Z 725.745,A -85,B 0,C 180,E1 17368.47,E2 17368.47} C_VEL
LIN {X 0,Y 373.133,Z 719.218,A -85,B 0,C 180,E1 17368.29,E2 17368.29} C_VEL
LIN {X 0,Y 374.338,Z 660.484,A -85,B 0,C 180,E1 17367.115,E2 17367.115} C_VEL
LIN {X 0,Y 369.15,Z 629.506,A -85,B 0,C 180,E1 17366.038,E2 17366.038} C_VEL
LIN {X 0,Y 372.134,Z 601.695,A -85,B 0,C 180,E1 17361.656,E2 17361.656} C_VEL
LIN {X 0,Y 374.811,Z 578.797,A -85,B 0,C 180,E1 17357.99,E2 17357.99} C_VEL
LIN {X 0,Y 370.516,Z 562.27,A -85,B 0,C 180,E1 17354.665,E2 17354.665} C_VEL
LIN {X 0,Y 365.871,Z 546.568,A -85,B 0,C 180,E1 17351.27,E2 17351.27} C_VEL
LIN {X 0,Y 361.747,Z 533.833,A -85,B 0,C 180,E1 17348.261,E2 17348.261} C_VEL
LIN {X 0,Y 361.731,Z 533.721,A -85,B 0,C 180,E1 17344.105,E2 17344.105} C_VEL
LIN {X 0,Y 361.723,Z 533.673,A -85,B 0,C 180,E1 17339.904,E2 17339.904} C_VEL
LIN {X 0,Y 361.733,Z 533.737,A -85,B 0,C 180,E1 17335.738,E2 17335.738} C_VEL
LIN {X 0,Y 361.734,Z 533.729,A -85,B 0,C 180,E1 17331.545,E2 17331.545} C_VEL
LIN {X 0,Y 361.732,Z 533.714,A -85,B 0,C 180,E1 17327.563,E2 17327.563} C_VEL
LIN {X 0,Y 361.738,Z 533.735,A -85,B 0,C 180,E1 17323.372,E2 17323.372} C_VEL
LIN {X 0,Y 361.738,Z 533.729,A -85,B 0,C 180,E1 17319.27,E2 17319.27} C_VEL
LIN {X 0,Y 361.74,Z 533.712,A -85,B 0,C 180,E1 17315.094,E2 17315.094} C_VEL
LIN {X 0,Y 361.745,Z 533.733,A -85,B 0,C 180,E1 17310.938,E2 17310.938} C_VEL
LIN {X 0,Y 361.743,Z 533.705,A -85,B 0,C 180,E1 17306.956,E2 17306.956} C_VEL
LIN {X 0,Y 361.748,Z 533.732,A -85,B 0,C 180,E1 17302.766,E2 17302.766} C_VEL
LIN {X 0,Y 361.748,Z 533.704,A -85,B 0,C 180,E1 17298.701,E2 17298.701} C_VEL
LIN {X 0,Y 361.748,Z 533.729,A -85,B 0,C 180,E1 17294.568,E2 17294.568} C_VEL
LIN {X 0,Y 361.75,Z 533.712,A -85,B 0,C 180,E1 17290.511,E2 17290.511} C_VEL
LIN {X 0,Y 361.754,Z 533.723,A -85,B 0,C 180,E1 17286.348,E2 17286.348} C_VEL
LIN {X 0,Y 361.754,Z 533.716,A -85,B 0,C 180,E1 17282.218,E2 17282.218} C_VEL
LIN {X 0,Y 361.757,Z 533.724,A -85,B 0,C 180,E1 17278.1,E2 17278.1} C_VEL
LIN {X 0,Y 361.758,Z 533.717,A -85,B 0,C 180,E1 17273.972,E2 17273.972} C_VEL
LIN {X 0,Y 361.762,Z 533.729,A -85,B 0,C 180,E1 17269.812,E2 17269.812} C_VEL
LIN {X 0,Y 361.761,Z 533.707,A -85,B 0,C 180,E1 17265.597,E2 17265.597} C_VEL
LIN {X 0,Y 361.768,Z 533.734,A -85,B 0,C 180,E1 17261.43,E2 17261.43} C_VEL
LIN {X 0,Y 361.766,Z 533.725,A -85,B 0,C 180,E1 17257.379,E2 17257.379} C_VEL
LIN {X 0,Y 361.77,Z 533.712,A -85,B 0,C 180,E1 17253.21,E2 17253.21} C_VEL
LIN {X 0,Y 361.772,Z 533.718,A -85,B 0,C 180,E1 17249.065,E2 17249.065} C_VEL
LIN {X 0,Y 361.773,Z 533.72,A -85,B 0,C 180,E1 17244.889,E2 17244.889} C_VEL
LIN {X 0,Y 361.775,Z 533.721,A -85,B 0,C 180,E1 17240.736,E2 17240.736} C_VEL
LIN {X 0,Y 361.804,Z 533.939,A -85,B 0,C 180,E1 17236.836,E2 17236.836} C_VEL
LIN {X 0,Y 368.203,Z 551.001,A -85,B 0,C 180,E1 17233.528,E2 17233.528} C_VEL
LIN {X 0,Y 374.841,Z 569.763,A -85,B 0,C 180,E1 17230.281,E2 17230.281} C_VEL
LIN {X 0,Y 380.381,Z 587.32,A -85,B 0,C 180,E1 17227.523,E2 17227.523} C_VEL
LIN {X 0,Y 376.355,Z 618.009,A -85,B 0,C 180,E1 17224.162,E2 17224.162} C_VEL
LIN {X 0,Y 379.185,Z 647.186,A -85,B 0,C 180,E1 17223.342,E2 17223.342} C_VEL
LIN {X 0,Y 375.587,Z 812.014,A -85,B 0,C 180,E1 17220.235,E2 17220.235} C_VEL
LIN {X 0,Y 374.487,Z 830.579,A -85,B 0,C 180,E1 17219.621,E2 17219.621} C_VEL
LIN {X 0,Y 372.925,Z 848.904,A -85,B 0,C 180,E1 17218.727,E2 17218.727} C_VEL
LIN {X 0,Y 371.158,Z 866.128,A -85,B 0,C 180,E1 17217.59,E2 17217.59} C_VEL
LIN {X 0,Y 369.267,Z 882.648,A -85,B 0,C 180,E1 17216.19,E2 17216.19} C_VEL
LIN {X 0,Y 367.265,Z 898.385,A -85,B 0,C 180,E1 17214.53,E2 17214.53} C_VEL
LIN {X 0,Y 365.413,Z 913.187,A -85,B 0,C 180,E1 17212.609,E2 17212.609} C_VEL
LIN {X 0,Y 363.726,Z 926.892,A -85,B 0,C 180,E1 17210.433,E2 17210.433} C_VEL
LIN {X 0,Y 362.406,Z 938.665,A -85,B 0,C 180,E1 17208.166,E2 17208.166} C_VEL
LIN {X 0,Y 361.456,Z 949.156,A -85,B 0,C 180,E1 17205.712,E2 17205.712} C_VEL
LIN {X 0,Y 360.891,Z 958.116,A -85,B 0,C 180,E1 17203.132,E2 17203.132} C_VEL
LIN {X 0,Y 360.705,Z 965.659,A -85,B 0,C 180,E1 17200.381,E2 17200.381} C_VEL
LIN {X 0,Y 360.791,Z 971.312,A -85,B 0,C 180,E1 17197.646,E2 17197.646} C_VEL
LIN {X 0,Y 361.032,Z 975.221,A -85,B 0,C 180,E1 17194.927,E2 17194.927} C_VEL
LIN {X 0,Y 361.239,Z 977.457,A -85,B 0,C 180,E1 17192.223,E2 17192.223} C_VEL
LIN {X 0,Y 361.295,Z 978.089,A -85,B 0,C 180,E1 17189.685,E2 17189.685} C_VEL
LIN {X 0,Y 361.164,Z 977.152,A -85,B 0,C 180,E1 17186.987,E2 17186.987} C_VEL
LIN {X 0,Y 360.916,Z 974.586,A -85,B 0,C 180,E1 17184.279,E2 17184.279} C_VEL
LIN {X 0,Y 360.681,Z 970.103,A -85,B 0,C 180,E1 17181.393,E2 17181.393} C_VEL
LIN {X 0,Y 360.677,Z 963.693,A -85,B 0,C 180,E1 17178.49,E2 17178.49} C_VEL
LIN {X 0,Y 361.042,Z 955.718,A -85,B 0,C 180,E1 17175.734,E2 17175.734} C_VEL
LIN {X 0,Y 361.834,Z 946.321,A -85,B 0,C 180,E1 17173.137,E2 17173.137} C_VEL
LIN {X 0,Y 363.144,Z 934.767,A -85,B 0,C 180,E1 17170.544,E2 17170.544} C_VEL
LIN {X 0,Y 364.922,Z 921.574,A -85,B 0,C 180,E1 17168.126,E2 17168.126} C_VEL
LIN {X 0,Y 366.896,Z 907.762,A -85,B 0,C 180,E1 17166.047,E2 17166.047} C_VEL
LIN {X 0,Y 369.07,Z 893.119,A -85,B 0,C 180,E1 17164.231,E2 17164.231} C_VEL
LIN {X 0,Y 371.391,Z 876.856,A -85,B 0,C 180,E1 17162.594,E2 17162.594} C_VEL
LIN {X 0,Y 373.501,Z 860.513,A -85,B 0,C 180,E1 17161.286,E2 17161.286} C_VEL
LIN {X 0,Y 375.521,Z 842.688,A -85,B 0,C 180,E1 17160.192,E2 17160.192} C_VEL
LIN {X 0,Y 377.144,Z 824.708,A -85,B 0,C 180,E1 17159.396,E2 17159.396} C_VEL
LIN {X 0,Y 378.206,Z 806.133,A -85,B 0,C 180,E1 17158.853,E2 17158.853} C_VEL
LIN {X 0,Y 382.153,Z 644.615,A -85,B 0,C 180,E1 17155.736,E2 17155.736} C_VEL
LIN {X 0,Y 379.325,Z 618.002,A -85,B 0,C 180,E1 17154.815,E2 17154.815} C_VEL
LIN {X 0,Y 383.668,Z 590.767,A -85,B 0,C 180,E1 17151.667,E2 17151.667} C_VEL
LIN {X 0,Y 379.15,Z 576.449,A -85,B 0,C 180,E1 17149.072,E2 17149.072} C_VEL
LIN {X 0,Y 374.051,Z 562.513,A -85,B 0,C 180,E1 17146.197,E2 17146.197} C_VEL
LIN {X 0,Y 368.901,Z 549.809,A -85,B 0,C 180,E1 17143.198,E2 17143.198} C_VEL
LIN {X 0,Y 364.962,Z 541.268,A -85,B 0,C 180,E1 17140.884,E2 17140.884} C_VEL
LIN {X 0,Y 363.098,Z 537.232,A -85,B 0,C 180,E1 17139.706,E2 17139.706} C_VEL
LIN {X 0,Y 361.795,Z 533.887,A -85,B 0,C 180,E1 17138.651,E2 17138.651} C_VEL
LIN {X 0,Y 361.769,Z 533.725,A -85,B 0,C 180,E1 17134.512,E2 17134.512} C_VEL
LIN {X 0,Y 361.768,Z 533.732,A -85,B 0,C 180,E1 17130.383,E2 17130.383} C_VEL
LIN {X 0,Y 361.756,Z 533.732,A -85,B 0,C 180,E1 17126.422,E2 17126.422} C_VEL
LIN {X 0,Y 361.746,Z 533.727,A -85,B 0,C 180,E1 17122.422,E2 17122.422} C_VEL
LIN {X 0,Y 361.74,Z 533.719,A -85,B 0,C 180,E1 17118.367,E2 17118.367} C_VEL
LIN {X 0,Y 361.734,Z 533.712,A -85,B 0,C 180,E1 17114.241,E2 17114.241} C_VEL
LIN {X 0,Y 361.729,Z 533.718,A -85,B 0,C 180,E1 17110.189,E2 17110.189} C_VEL
LIN {X 0,Y 361.733,Z 533.731,A -85,B 0,C 180,E1 17106.188,E2 17106.188} C_VEL
LIN {X 0,Y 361.741,Z 533.737,A -85,B 0,C 180,E1 17102.059,E2 17102.059} C_VEL
LIN {X 0,Y 361.746,Z 533.734,A -85,B 0,C 180,E1 17097.94,E2 17097.94} C_VEL
LIN {X 0,Y 361.749,Z 533.724,A -85,B 0,C 180,E1 17093.811,E2 17093.811} C_VEL
LIN {X 0,Y 361.755,Z 533.72,A -85,B 0,C 180,E1 17089.65,E2 17089.65} C_VEL
LIN {X 0,Y 361.758,Z 533.72,A -85,B 0,C 180,E1 17085.596,E2 17085.596} C_VEL
LIN {X 0,Y 361.764,Z 533.726,A -85,B 0,C 180,E1 17081.42,E2 17081.42} C_VEL
LIN {X 0,Y 361.768,Z 533.737,A -85,B 0,C 180,E1 17077.368,E2 17077.368} C_VEL
LIN {X 0,Y 361.872,Z 534.137,A -85,B 0,C 180,E1 17076.468,E2 17076.468} C_VEL
LIN {X 0,Y 366.376,Z 545.37,A -85,B 0,C 180,E1 17072.818,E2 17072.818} C_VEL
LIN {X 0,Y 370.57,Z 556.9,A -85,B 0,C 180,E1 17069.518,E2 17069.518} C_VEL
LIN {X 0,Y 374.546,Z 569.551,A -85,B 0,C 180,E1 17066.271,E2 17066.271} C_VEL
LIN {X 0,Y 377.914,Z 582.504,A -85,B 0,C 180,E1 17063.277,E2 17063.277} C_VEL
LIN {X 0,Y 378.526,Z 585.745,A -85,B 0,C 180,E1 17062.588,E2 17062.588} C_VEL
LIN {X 0,Y 374.453,Z 612.784,A -85,B 0,C 180,E1 17058.121,E2 17058.121} C_VEL
LIN {X 0,Y 372.323,Z 629.33,A -85,B 0,C 180,E1 17055.44,E2 17055.44} C_VEL
LIN {X 0,Y 373.759,Z 636.616,A -85,B 0,C 180,E1 17055.056,E2 17055.056} C_VEL
LIN {X 0,Y 378.766,Z 663.47,A -85,B 0,C 180,E1 17053.932,E2 17053.932} C_VEL
LIN {X 0,Y 375.919,Z 757.648,A -85,B 0,C 180,E1 17051.942,E2 17051.942} C_VEL
LIN {X 0,Y 375.171,Z 773.603,A -85,B 0,C 180,E1 17051.326,E2 17051.326} C_VEL
LIN {X 0,Y 374.105,Z 788.183,A -85,B 0,C 180,E1 17050.494,E2 17050.494} C_VEL
LIN {X 0,Y 372.624,Z 802.75,A -85,B 0,C 180,E1 17049.35,E2 17049.35} C_VEL
LIN {X 0,Y 370.969,Z 815.862,A -85,B 0,C 180,E1 17048.009,E2 17048.009} C_VEL
LIN {X 0,Y 369.161,Z 828.27,A -85,B 0,C 180,E1 17046.375,E2 17046.375} C_VEL
LIN {X 0,Y 367.441,Z 838.928,A -85,B 0,C 180,E1 17044.586,E2 17044.586} C_VEL
LIN {X 0,Y 365.808,Z 848.369,A -85,B 0,C 180,E1 17042.573,E2 17042.573} C_VEL
LIN {X 0,Y 364.436,Z 855.877,A -85,B 0,C 180,E1 17040.496,E2 17040.496} C_VEL
LIN {X 0,Y 363.322,Z 862.011,A -85,B 0,C 180,E1 17038.247,E2 17038.247} C_VEL
LIN {X 0,Y 362.488,Z 866.585,A -85,B 0,C 180,E1 17035.833,E2 17035.833} C_VEL
LIN {X 0,Y 361.944,Z 869.497,A -85,B 0,C 180,E1 17033.264,E2 17033.264} C_VEL
LIN {X 0,Y 361.676,Z 870.453,A -85,B 0,C 180,E1 17030.72,E2 17030.72} C_VEL
LIN {X 0,Y 361.651,Z 869.658,A -85,B 0,C 180,E1 17028.201,E2 17028.201} C_VEL
LIN {X 0,Y 361.884,Z 866.838,A -85,B 0,C 180,E1 17025.542,E2 17025.542} C_VEL
LIN {X 0,Y 362.359,Z 862.268,A -85,B 0,C 180,E1 17023.083,E2 17023.083} C_VEL
LIN {X 0,Y 363.092,Z 856.171,A -85,B 0,C 180,E1 17020.79,E2 17020.79} C_VEL
LIN {X 0,Y 364.141,Z 847.979,A -85,B 0,C 180,E1 17018.524,E2 17018.524} C_VEL
LIN {X 0,Y 365.343,Z 838.778,A -85,B 0,C 180,E1 17016.558,E2 17016.558} C_VEL
LIN {X 0,Y 366.744,Z 827.648,A -85,B 0,C 180,E1 17014.689,E2 17014.689} C_VEL
LIN {X 0,Y 368.105,Z 815.692,A -85,B 0,C 180,E1 17013.112,E2 17013.112} C_VEL
LIN {X 0,Y 369.513,Z 802.085,A -85,B 0,C 180,E1 17011.704,E2 17011.704} C_VEL
LIN {X 0,Y 370.737,Z 787.177,A -85,B 0,C 180,E1 17010.539,E2 17010.539} C_VEL
LIN {X 0,Y 371.658,Z 772.119,A -85,B 0,C 180,E1 17009.685,E2 17009.685} C_VEL
LIN {X 0,Y 372.285,Z 755.917,A -85,B 0,C 180,E1 17009.075,E2 17009.075} C_VEL
LIN {X 0,Y 373.133,Z 719.218,A -85,B 0,C 180,E1 17008.29,E2 17008.29} C_VEL
LIN {X 0,Y 372.367,Z 711.617,A -85,B 0,C 180,E1 17008.07,E2 17008.07} C_VEL
LIN {X 0,Y 367.156,Z 691.67,A -85,B 0,C 180,E1 17007.274,E2 17007.274} C_VEL
LIN {X 0,Y 366.665,Z 685.131,A -85,B 0,C 180,E1 17007.098,E2 17007.098} C_VEL
LIN {X 0,Y 367.038,Z 661.474,A -85,B 0,C 180,E1 17006.611,E2 17006.611} C_VEL
LIN {X 0,Y 361.71,Z 629.457,A -85,B 0,C 180,E1 17005.48,E2 17005.48} C_VEL
LIN {X 0,Y 364.872,Z 601.584,A -85,B 0,C 180,E1 17001.013,E2 17001.013} C_VEL
LIN {X 0,Y 367.366,Z 581.289,A -85,B 0,C 180,E1 16997.714,E2 16997.714} C_VEL
LIN {X 0,Y 363.135,Z 564.898,A -85,B 0,C 180,E1 16994.345,E2 16994.345} C_VEL
LIN {X 0,Y 358.594,Z 549.523,A -85,B 0,C 180,E1 16990.95,E2 16990.95} C_VEL
LIN {X 0,Y 354.167,Z 536.28,A -85,B 0,C 180,E1 16987.819,E2 16987.819} C_VEL
LIN {X 0,Y 353.848,Z 534.834,A -85,B 0,C 180,E1 16987.4,E2 16987.4} C_VEL
LIN {X 0,Y 353.831,Z 534.724,A -85,B 0,C 180,E1 16983.248,E2 16983.248} C_VEL
LIN {X 0,Y 353.828,Z 534.654,A -85,B 0,C 180,E1 16979.05,E2 16979.05} C_VEL
LIN {X 0,Y 353.831,Z 534.722,A -85,B 0,C 180,E1 16974.799,E2 16974.799} C_VEL
LIN {X 0,Y 353.832,Z 534.724,A -85,B 0,C 180,E1 16970.522,E2 16970.522} C_VEL
LIN {X 0,Y 353.826,Z 534.704,A -85,B 0,C 180,E1 16966.338,E2 16966.338} C_VEL
LIN {X 0,Y 353.831,Z 534.7,A -85,B 0,C 180,E1 16962.24,E2 16962.24} C_VEL
LIN {X 0,Y 353.829,Z 534.725,A -85,B 0,C 180,E1 16958.027,E2 16958.027} C_VEL
LIN {X 0,Y 353.821,Z 534.689,A -85,B 0,C 180,E1 16953.822,E2 16953.822} C_VEL
LIN {X 0,Y 353.837,Z 534.721,A -85,B 0,C 180,E1 16949.824,E2 16949.824} C_VEL
LIN {X 0,Y 353.83,Z 534.684,A -85,B 0,C 180,E1 16945.659,E2 16945.659} C_VEL
LIN {X 0,Y 353.84,Z 534.72,A -85,B 0,C 180,E1 16941.552,E2 16941.552} C_VEL
LIN {X 0,Y 353.836,Z 534.68,A -85,B 0,C 180,E1 16937.43,E2 16937.43} C_VEL
LIN {X 0,Y 353.85,Z 534.721,A -85,B 0,C 180,E1 16933.398,E2 16933.398} C_VEL
LIN {X 0,Y 353.844,Z 534.676,A -85,B 0,C 180,E1 16929.269,E2 16929.269} C_VEL
LIN {X 0,Y 353.852,Z 534.718,A -85,B 0,C 180,E1 16925.188,E2 16925.188} C_VEL
LIN {X 0,Y 353.848,Z 534.678,A -85,B 0,C 180,E1 16920.972,E2 16920.972} C_VEL
LIN {X 0,Y 353.845,Z 534.721,A -85,B 0,C 180,E1 16916.761,E2 16916.761} C_VEL
LIN {X 0,Y 353.846,Z 534.684,A -85,B 0,C 180,E1 16912.642,E2 16912.642} C_VEL
LIN {X 0,Y 353.845,Z 534.72,A -85,B 0,C 180,E1 16908.427,E2 16908.427} C_VEL
LIN {X 0,Y 353.843,Z 534.697,A -85,B 0,C 180,E1 16904.261,E2 16904.261} C_VEL
LIN {X 0,Y 353.848,Z 534.707,A -85,B 0,C 180,E1 16900.179,E2 16900.179} C_VEL
LIN {X 0,Y 353.857,Z 534.72,A -85,B 0,C 180,E1 16896.168,E2 16896.168} C_VEL
LIN {X 0,Y 353.86,Z 534.709,A -85,B 0,C 180,E1 16892.028,E2 16892.028} C_VEL
LIN {X 0,Y 353.858,Z 534.705,A -85,B 0,C 180,E1 16887.913,E2 16887.913} C_VEL
LIN {X 0,Y 353.858,Z 534.708,A -85,B 0,C 180,E1 16883.804,E2 16883.804} C_VEL
LIN {X 0,Y 353.869,Z 534.716,A -85,B 0,C 180,E1 16879.681,E2 16879.681} C_VEL
LIN {X 0,Y 353.91,Z 535.016,A -85,B 0,C 180,E1 16877.717,E2 16877.717} C_VEL
LIN {X 0,Y 360.834,Z 553.306,A -85,B 0,C 180,E1 16874.066,E2 16874.066} C_VEL
LIN {X 0,Y 367.588,Z 572.618,A -85,B 0,C 180,E1 16870.633,E2 16870.633} C_VEL
LIN {X 0,Y 373.034,Z 589.494,A -85,B 0,C 180,E1 16867.912,E2 16867.912} C_VEL
LIN {X 0,Y 369.085,Z 617.952,A -85,B 0,C 180,E1 16864.719,E2 16864.719} C_VEL
LIN {X 0,Y 371.922,Z 648.057,A -85,B 0,C 180,E1 16863.845,E2 16863.845} C_VEL
LIN {X 0,Y 368.187,Z 811.459,A -85,B 0,C 180,E1 16860.71,E2 16860.71} C_VEL
LIN {X 0,Y 367.067,Z 829.914,A -85,B 0,C 180,E1 16860.09,E2 16860.09} C_VEL
LIN {X 0,Y 365.469,Z 847.981,A -85,B 0,C 180,E1 16859.197,E2 16859.197} C_VEL
LIN {X 0,Y 363.641,Z 865.25,A -85,B 0,C 180,E1 16858.041,E2 16858.041} C_VEL
LIN {X 0,Y 361.66,Z 881.904,A -85,B 0,C 180,E1 16856.607,E2 16856.607} C_VEL
LIN {X 0,Y 359.58,Z 897.616,A -85,B 0,C 180,E1 16854.914,E2 16854.914} C_VEL
LIN {X 0,Y 357.645,Z 912.382,A -85,B 0,C 180,E1 16852.954,E2 16852.954} C_VEL
LIN {X 0,Y 355.884,Z 926.042,A -85,B 0,C 180,E1 16850.732,E2 16850.732} C_VEL
LIN {X 0,Y 354.505,Z 937.78,A -85,B 0,C 180,E1 16848.415,E2 16848.415} C_VEL
LIN {X 0,Y 353.517,Z 948.172,A -85,B 0,C 180,E1 16845.924,E2 16845.924} C_VEL
LIN {X 0,Y 352.928,Z 957.161,A -85,B 0,C 180,E1 16843.267,E2 16843.267} C_VEL
LIN {X 0,Y 352.743,Z 964.795,A -85,B 0,C 180,E1 16840.398,E2 16840.398} C_VEL
LIN {X 0,Y 352.858,Z 970.56,A -85,B 0,C 180,E1 16837.491,E2 16837.491} C_VEL
LIN {X 0,Y 353.128,Z 974.348,A -85,B 0,C 180,E1 16834.683,E2 16834.683} C_VEL
LIN {X 0,Y 353.345,Z 976.394,A -85,B 0,C 180,E1 16831.948,E2 16831.948} C_VEL
LIN {X 0,Y 353.378,Z 976.825,A -85,B 0,C 180,E1 16829.191,E2 16829.191} C_VEL
LIN {X 0,Y 353.197,Z 975.626,A -85,B 0,C 180,E1 16826.432,E2 16826.432} C_VEL
LIN {X 0,Y 352.903,Z 972.805,A -85,B 0,C 180,E1 16823.659,E2 16823.659} C_VEL
LIN {X 0,Y 352.693,Z 968.331,A -85,B 0,C 180,E1 16820.868,E2 16820.868} C_VEL
LIN {X 0,Y 352.725,Z 961.821,A -85,B 0,C 180,E1 16817.948,E2 16817.948} C_VEL
LIN {X 0,Y 353.195,Z 953.48,A -85,B 0,C 180,E1 16815.075,E2 16815.075} C_VEL
LIN {X 0,Y 354.194,Z 943.16,A -85,B 0,C 180,E1 16812.253,E2 16812.253} C_VEL
LIN {X 0,Y 355.614,Z 931.999,A -85,B 0,C 180,E1 16809.771,E2 16809.771} C_VEL
LIN {X 0,Y 357.448,Z 919.49,A -85,B 0,C 180,E1 16807.471,E2 16807.471} C_VEL
LIN {X 0,Y 359.59,Z 905.531,A -85,B 0,C 180,E1 16805.354,E2 16805.354} C_VEL
LIN {X 0,Y 361.913,Z 890.779,A -85,B 0,C 180,E1 16803.523,E2 16803.523} C_VEL
LIN {X 0,Y 364.283,Z 874.875,A -85,B 0,C 180,E1 16801.924,E2 16801.924} C_VEL
LIN {X 0,Y 366.521,Z 858.198,A -85,B 0,C 180,E1 16800.596,E2 16800.596} C_VEL
LIN {X 0,Y 368.594,Z 840.519,A -85,B 0,C 180,E1 16799.524,E2 16799.524} C_VEL
LIN {X 0,Y 370.257,Z 822.494,A -85,B 0,C 180,E1 16798.737,E2 16798.737} C_VEL
LIN {X 0,Y 371.321,Z 803.191,A -85,B 0,C 180,E1 16798.19,E2 16798.19} C_VEL
LIN {X 0,Y 375.41,Z 645.606,A -85,B 0,C 180,E1 16795.097,E2 16795.097} C_VEL
LIN {X 0,Y 372.536,Z 618.147,A -85,B 0,C 180,E1 16794.115,E2 16794.115} C_VEL
LIN {X 0,Y 376.625,Z 593.594,A -85,B 0,C 180,E1 16791.212,E2 16791.212} C_VEL
LIN {X 0,Y 371.925,Z 578.615,A -85,B 0,C 180,E1 16788.4,E2 16788.4} C_VEL
LIN {X 0,Y 366.73,Z 564.519,A -85,B 0,C 180,E1 16785.365,E2 16785.365} C_VEL
LIN {X 0,Y 361.274,Z 551.264,A -85,B 0,C 180,E1 16782.048,E2 16782.048} C_VEL
LIN {X 0,Y 357.129,Z 542.391,A -85,B 0,C 180,E1 16779.459,E2 16779.459} C_VEL
LIN {X 0,Y 355.357,Z 538.464,A -85,B 0,C 180,E1 16778.244,E2 16778.244} C_VEL
LIN {X 0,Y 353.844,Z 534.878,A -85,B 0,C 180,E1 16777.004,E2 16777.004} C_VEL
LIN {X 0,Y 353.817,Z 534.713,A -85,B 0,C 180,E1 16772.859,E2 16772.859} C_VEL
LIN {X 0,Y 353.813,Z 534.709,A -85,B 0,C 180,E1 16768.712,E2 16768.712} C_VEL
LIN {X 0,Y 353.808,Z 534.708,A -85,B 0,C 180,E1 16764.515,E2 16764.515} C_VEL
LIN {X 0,Y 353.802,Z 534.715,A -85,B 0,C 180,E1 16760.513,E2 16760.513} C_VEL
LIN {X 0,Y 353.799,Z 534.727,A -85,B 0,C 180,E1 16756.416,E2 16756.416} C_VEL
LIN {X 0,Y 353.796,Z 534.727,A -85,B 0,C 180,E1 16752.237,E2 16752.237} C_VEL
LIN {X 0,Y 353.793,Z 534.716,A -85,B 0,C 180,E1 16748.123,E2 16748.123} C_VEL
LIN {X 0,Y 353.797,Z 534.703,A -85,B 0,C 180,E1 16744.051,E2 16744.051} C_VEL
LIN {X 0,Y 353.799,Z 534.702,A -85,B 0,C 180,E1 16740,E2 16740} C_VEL
LIN {X 0,Y 353.808,Z 534.706,A -85,B 0,C 180,E1 16735.786,E2 16735.786} C_VEL
LIN {X 0,Y 353.813,Z 534.713,A -85,B 0,C 180,E1 16731.713,E2 16731.713} C_VEL
LIN {X 0,Y 353.819,Z 534.715,A -85,B 0,C 180,E1 16727.598,E2 16727.598} C_VEL
LIN {X 0,Y 353.825,Z 534.712,A -85,B 0,C 180,E1 16723.416,E2 16723.416} C_VEL
LIN {X 0,Y 353.83,Z 534.709,A -85,B 0,C 180,E1 16719.265,E2 16719.265} C_VEL
LIN {X 0,Y 353.902,Z 535.064,A -85,B 0,C 180,E1 16718.103,E2 16718.103} C_VEL
LIN {X 0,Y 357.257,Z 543.3,A -85,B 0,C 180,E1 16715.177,E2 16715.177} C_VEL
LIN {X 0,Y 361.129,Z 553.236,A -85,B 0,C 180,E1 16712.019,E2 16712.019} C_VEL
LIN {X 0,Y 365.208,Z 565.159,A -85,B 0,C 180,E1 16708.655,E2 16708.655} C_VEL
LIN {X 0,Y 368.884,Z 577.717,A -85,B 0,C 180,E1 16705.476,E2 16705.476} C_VEL
LIN {X 0,Y 371.442,Z 588.637,A -85,B 0,C 180,E1 16702.97,E2 16702.97} C_VEL
LIN {X 0,Y 367.195,Z 615.343,A -85,B 0,C 180,E1 16698.479,E2 16698.479} C_VEL
LIN {X 0,Y 365.315,Z 629.43,A -85,B 0,C 180,E1 16696.175,E2 16696.175} C_VEL
LIN {X 0,Y 370.586,Z 655.931,A -85,B 0,C 180,E1 16694.935,E2 16694.935} C_VEL
LIN {X 0,Y 372.01,Z 665.566,A -85,B 0,C 180,E1 16694.562,E2 16694.562} C_VEL
LIN {X 0,Y 369.043,Z 758.267,A -85,B 0,C 180,E1 16692.564,E2 16692.564} C_VEL
LIN {X 0,Y 368.248,Z 774.249,A -85,B 0,C 180,E1 16691.937,E2 16691.937} C_VEL
LIN {X 0,Y 367.115,Z 788.896,A -85,B 0,C 180,E1 16691.087,E2 16691.087} C_VEL
LIN {X 0,Y 365.509,Z 803.787,A -85,B 0,C 180,E1 16689.896,E2 16689.896} C_VEL
LIN {X 0,Y 363.75,Z 816.914,A -85,B 0,C 180,E1 16688.523,E2 16688.523} C_VEL
LIN {X 0,Y 361.815,Z 829.447,A -85,B 0,C 180,E1 16686.84,E2 16686.84} C_VEL
LIN {X 0,Y 360.054,Z 839.743,A -85,B 0,C 180,E1 16685.082,E2 16685.082} C_VEL
LIN {X 0,Y 358.254,Z 849.497,A -85,B 0,C 180,E1 16682.967,E2 16682.967} C_VEL
LIN {X 0,Y 356.787,Z 857.003,A -85,B 0,C 180,E1 16680.848,E2 16680.848} C_VEL
LIN {X 0,Y 355.509,Z 863.55,A -85,B 0,C 180,E1 16678.374,E2 16678.374} C_VEL
LIN {X 0,Y 354.624,Z 867.985,A -85,B 0,C 180,E1 16675.909,E2 16675.909} C_VEL
LIN {X 0,Y 354.065,Z 870.708,A -85,B 0,C 180,E1 16673.395,E2 16673.395} C_VEL
LIN {X 0,Y 353.764,Z 871.652,A -85,B 0,C 180,E1 16670.685,E2 16670.685} C_VEL
LIN {X 0,Y 353.737,Z 870.757,A -85,B 0,C 180,E1 16668.111,E2 16668.111} C_VEL
LIN {X 0,Y 353.963,Z 868.096,A -85,B 0,C 180,E1 16665.563,E2 16665.563} C_VEL
LIN {X 0,Y 354.415,Z 863.937,A -85,B 0,C 180,E1 16663.206,E2 16663.206} C_VEL
LIN {X 0,Y 355.212,Z 857.553,A -85,B 0,C 180,E1 16660.704,E2 16660.704} C_VEL
LIN {X 0,Y 356.209,Z 850.096,A -85,B 0,C 180,E1 16658.553,E2 16658.553} C_VEL
LIN {X 0,Y 357.517,Z 840.584,A -85,B 0,C 180,E1 16656.42,E2 16656.42} C_VEL
LIN {X 0,Y 359.025,Z 829.097,A -85,B 0,C 180,E1 16654.43,E2 16654.43} C_VEL
LIN {X 0,Y 360.407,Z 817.625,A -85,B 0,C 180,E1 16652.86,E2 16652.86} C_VEL
LIN {X 0,Y 361.857,Z 804.268,A -85,B 0,C 180,E1 16651.423,E2 16651.423} C_VEL
LIN {X 0,Y 363.133,Z 789.822,A -85,B 0,C 180,E1 16650.235,E2 16650.235} C_VEL
LIN {X 0,Y 364.145,Z 774.94,A -85,B 0,C 180,E1 16649.33,E2 16649.33} C_VEL
LIN {X 0,Y 364.842,Z 758.449,A -85,B 0,C 180,E1 16648.663,E2 16648.663} C_VEL
LIN {X 0,Y 366.138,Z 705.883,A -85,B 0,C 180,E1 16647.519,E2 16647.519} C_VEL
LIN {X 0,Y 366.665,Z 685.131,A -85,B 0,C 180,E1 16647.098,E2 16647.098} C_VEL
LIN {X 0,Y 365.941,Z 677.503,A -85,B 0,C 180,E1 16646.879,E2 16646.879} C_VEL
LIN {X 0,Y 362.811,Z 667.115,A -85,B 0,C 180,E1 16646.419,E2 16646.419} C_VEL
LIN {X 0,Y 358.644,Z 654.662,A -85,B 0,C 180,E1 16645.825,E2 16645.825} C_VEL
LIN {X 0,Y 357.953,Z 651.42,A -85,B 0,C 180,E1 16645.7,E2 16645.7} C_VEL
LIN {X 0,Y 354.295,Z 629.342,A -85,B 0,C 180,E1 16644.89,E2 16644.89} C_VEL
LIN {X 0,Y 357.637,Z 601.419,A -85,B 0,C 180,E1 16640.342,E2 16640.342} C_VEL
LIN {X 0,Y 359.905,Z 583.665,A -85,B 0,C 180,E1 16637.403,E2 16637.403} C_VEL
LIN {X 0,Y 355.567,Z 566.702,A -85,B 0,C 180,E1 16633.835,E2 16633.835} C_VEL
LIN {X 0,Y 350.879,Z 550.98,A -85,B 0,C 180,E1 16630.264,E2 16630.264} C_VEL
LIN {X 0,Y 346.418,Z 537.693,A -85,B 0,C 180,E1 16627.033,E2 16627.033} C_VEL
LIN {X 0,Y 345.866,Z 535.765,A -85,B 0,C 180,E1 16626.408,E2 16626.408} C_VEL
LIN {X 0,Y 345.854,Z 535.694,A -85,B 0,C 180,E1 16622.209,E2 16622.209} C_VEL
LIN {X 0,Y 345.845,Z 535.661,A -85,B 0,C 180,E1 16617.863,E2 16617.863} C_VEL
LIN {X 0,Y 345.854,Z 535.701,A -85,B 0,C 180,E1 16613.656,E2 16613.656} C_VEL
LIN {X 0,Y 345.86,Z 535.715,A -85,B 0,C 180,E1 16609.493,E2 16609.493} C_VEL
LIN {X 0,Y 345.863,Z 535.711,A -85,B 0,C 180,E1 16605.33,E2 16605.33} C_VEL
LIN {X 0,Y 345.859,Z 535.684,A -85,B 0,C 180,E1 16601.235,E2 16601.235} C_VEL
LIN {X 0,Y 345.867,Z 535.714,A -85,B 0,C 180,E1 16597.075,E2 16597.075} C_VEL
LIN {X 0,Y 345.865,Z 535.686,A -85,B 0,C 180,E1 16592.922,E2 16592.922} C_VEL
LIN {X 0,Y 345.869,Z 535.709,A -85,B 0,C 180,E1 16588.85,E2 16588.85} C_VEL
LIN {X 0,Y 345.873,Z 535.687,A -85,B 0,C 180,E1 16584.6,E2 16584.6} C_VEL
LIN {X 0,Y 345.876,Z 535.706,A -85,B 0,C 180,E1 16580.475,E2 16580.475} C_VEL
LIN {X 0,Y 345.876,Z 535.68,A -85,B 0,C 180,E1 16576.285,E2 16576.285} C_VEL
LIN {X 0,Y 345.882,Z 535.711,A -85,B 0,C 180,E1 16572.183,E2 16572.183} C_VEL
LIN {X 0,Y 345.882,Z 535.67,A -85,B 0,C 180,E1 16567.976,E2 16567.976} C_VEL
LIN {X 0,Y 345.89,Z 535.71,A -85,B 0,C 180,E1 16563.813,E2 16563.813} C_VEL
LIN {X 0,Y 345.887,Z 535.67,A -85,B 0,C 180,E1 16559.669,E2 16559.669} C_VEL
LIN {X 0,Y 345.895,Z 535.711,A -85,B 0,C 180,E1 16555.524,E2 16555.524} C_VEL
LIN {X 0,Y 345.888,Z 535.679,A -85,B 0,C 180,E1 16551.523,E2 16551.523} C_VEL
LIN {X 0,Y 345.896,Z 535.702,A -85,B 0,C 180,E1 16547.31,E2 16547.31} C_VEL
LIN {X 0,Y 345.899,Z 535.702,A -85,B 0,C 180,E1 16543.199,E2 16543.199} C_VEL
LIN {X 0,Y 345.902,Z 535.685,A -85,B 0,C 180,E1 16538.996,E2 16538.996} C_VEL
LIN {X 0,Y 345.909,Z 535.698,A -85,B 0,C 180,E1 16534.782,E2 16534.782} C_VEL
LIN {X 0,Y 345.92,Z 535.708,A -85,B 0,C 180,E1 16530.569,E2 16530.569} C_VEL
LIN {X 0,Y 345.923,Z 535.708,A -85,B 0,C 180,E1 16526.292,E2 16526.292} C_VEL
LIN {X 0,Y 345.933,Z 535.7,A -85,B 0,C 180,E1 16522.002,E2 16522.002} C_VEL
LIN {X 0,Y 345.937,Z 535.96,A -85,B 0,C 180,E1 16518.716,E2 16518.716} C_VEL
LIN {X 0,Y 352.366,Z 552.727,A -85,B 0,C 180,E1 16515.183,E2 16515.183} C_VEL
LIN {X 0,Y 358.991,Z 571.317,A -85,B 0,C 180,E1 16511.718,E2 16511.718} C_VEL
LIN {X 0,Y 365.632,Z 591.913,A -85,B 0,C 180,E1 16508.28,E2 16508.28} C_VEL
LIN {X 0,Y 361.833,Z 618.168,A -85,B 0,C 180,E1 16505.276,E2 16505.276} C_VEL
LIN {X 0,Y 364.693,Z 648.803,A -85,B 0,C 180,E1 16504.371,E2 16504.371} C_VEL
LIN {X 0,Y 360.813,Z 810.795,A -85,B 0,C 180,E1 16501.205,E2 16501.205} C_VEL
LIN {X 0,Y 359.661,Z 829.247,A -85,B 0,C 180,E1 16500.573,E2 16500.573} C_VEL
LIN {X 0,Y 358.037,Z 846.932,A -85,B 0,C 180,E1 16499.687,E2 16499.687} C_VEL
LIN {X 0,Y 356.137,Z 864.284,A -85,B 0,C 180,E1 16498.507,E2 16498.507} C_VEL
LIN {X 0,Y 354.069,Z 880.999,A -85,B 0,C 180,E1 16497.042,E2 16497.042} C_VEL
LIN {X 0,Y 351.911,Z 896.746,A -85,B 0,C 180,E1 16495.315,E2 16495.315} C_VEL
LIN {X 0,Y 349.89,Z 911.532,A -85,B 0,C 180,E1 16493.315,E2 16493.315} C_VEL
LIN {X 0,Y 348.054,Z 925.191,A -85,B 0,C 180,E1 16491.044,E2 16491.044} C_VEL
LIN {X 0,Y 346.611,Z 936.896,A -85,B 0,C 180,E1 16488.675,E2 16488.675} C_VEL
LIN {X 0,Y 345.578,Z 947.252,A -85,B 0,C 180,E1 16486.127,E2 16486.127} C_VEL
LIN {X 0,Y 344.966,Z 956.206,A -85,B 0,C 180,E1 16483.408,E2 16483.408} C_VEL
LIN {X 0,Y 344.781,Z 963.674,A -85,B 0,C 180,E1 16480.528,E2 16480.528} C_VEL
LIN {X 0,Y 344.903,Z 969.251,A -85,B 0,C 180,E1 16477.665,E2 16477.665} C_VEL
LIN {X 0,Y 345.192,Z 973.065,A -85,B 0,C 180,E1 16474.82,E2 16474.82} C_VEL
LIN {X 0,Y 345.428,Z 975.184,A -85,B 0,C 180,E1 16471.992,E2 16471.992} C_VEL
LIN {X 0,Y 345.467,Z 975.676,A -85,B 0,C 180,E1 16469.339,E2 16469.339} C_VEL
LIN {X 0,Y 345.275,Z 974.597,A -85,B 0,C 180,E1 16466.516,E2 16466.516} C_VEL
LIN {X 0,Y 344.954,Z 971.885,A -85,B 0,C 180,E1 16463.679,E2 16463.679} C_VEL
LIN {X 0,Y 344.713,Z 967.189,A -85,B 0,C 180,E1 16460.655,E2 16460.655} C_VEL
LIN {X 0,Y 344.749,Z 960.976,A -85,B 0,C 180,E1 16457.78,E2 16457.78} C_VEL
LIN {X 0,Y 345.236,Z 952.885,A -85,B 0,C 180,E1 16454.895,E2 16454.895} C_VEL
LIN {X 0,Y 346.206,Z 943.384,A -85,B 0,C 180,E1 16452.177,E2 16452.177} C_VEL
LIN {X 0,Y 347.78,Z 931.724,A -85,B 0,C 180,E1 16449.471,E2 16449.471} C_VEL
LIN {X 0,Y 349.704,Z 919.372,A -85,B 0,C 180,E1 16447.122,E2 16447.122} C_VEL
LIN {X 0,Y 351.947,Z 905.591,A -85,B 0,C 180,E1 16444.961,E2 16444.961} C_VEL
LIN {X 0,Y 354.429,Z 890.716,A -85,B 0,C 180,E1 16443.056,E2 16443.056} C_VEL
LIN {X 0,Y 356.968,Z 874.599,A -85,B 0,C 180,E1 16441.387,E2 16441.387} C_VEL
LIN {X 0,Y 359.303,Z 858.222,A -85,B 0,C 180,E1 16440.045,E2 16440.045} C_VEL
LIN {X 0,Y 361.477,Z 840.746,A -85,B 0,C 180,E1 16438.95,E2 16438.95} C_VEL
LIN {X 0,Y 363.245,Z 822.78,A -85,B 0,C 180,E1 16438.136,E2 16438.136} C_VEL
LIN {X 0,Y 364.374,Z 804.253,A -85,B 0,C 180,E1 16437.584,E2 16437.584} C_VEL
LIN {X 0,Y 368.719,Z 646.378,A -85,B 0,C 180,E1 16434.424,E2 16434.424} C_VEL
LIN {X 0,Y 365.804,Z 618.392,A -85,B 0,C 180,E1 16433.395,E2 16433.395} C_VEL
LIN {X 0,Y 369.676,Z 596.691,A -85,B 0,C 180,E1 16430.783,E2 16430.783} C_VEL
LIN {X 0,Y 365.21,Z 582.362,A -85,B 0,C 180,E1 16428.013,E2 16428.013} C_VEL
LIN {X 0,Y 360.32,Z 568.91,A -85,B 0,C 180,E1 16425.04,E2 16425.04} C_VEL
LIN {X 0,Y 355.123,Z 556.102,A -85,B 0,C 180,E1 16421.754,E2 16421.754} C_VEL
LIN {X 0,Y 351.157,Z 547.534,A -85,B 0,C 180,E1 16419.205,E2 16419.205} C_VEL
LIN {X 0,Y 349.131,Z 543.189,A -85,B 0,C 180,E1 16417.797,E2 16417.797} C_VEL
LIN {X 0,Y 347.461,Z 539.557,A -85,B 0,C 180,E1 16416.56,E2 16416.56} C_VEL
LIN {X 0,Y 345.898,Z 535.83,A -85,B 0,C 180,E1 16415.116,E2 16415.116} C_VEL
LIN {X 0,Y 345.876,Z 535.703,A -85,B 0,C 180,E1 16410.775,E2 16410.775} C_VEL
LIN {X 0,Y 345.873,Z 535.705,A -85,B 0,C 180,E1 16406.62,E2 16406.62} C_VEL
LIN {X 0,Y 345.868,Z 535.702,A -85,B 0,C 180,E1 16402.432,E2 16402.432} C_VEL
LIN {X 0,Y 345.868,Z 535.696,A -85,B 0,C 180,E1 16398.192,E2 16398.192} C_VEL
LIN {X 0,Y 345.862,Z 535.689,A -85,B 0,C 180,E1 16394.054,E2 16394.054} C_VEL
LIN {X 0,Y 345.857,Z 535.691,A -85,B 0,C 180,E1 16389.989,E2 16389.989} C_VEL
LIN {X 0,Y 345.858,Z 535.702,A -85,B 0,C 180,E1 16385.974,E2 16385.974} C_VEL
LIN {X 0,Y 345.868,Z 535.714,A -85,B 0,C 180,E1 16381.822,E2 16381.822} C_VEL
LIN {X 0,Y 345.874,Z 535.713,A -85,B 0,C 180,E1 16377.68,E2 16377.68} C_VEL
LIN {X 0,Y 345.881,Z 535.704,A -85,B 0,C 180,E1 16373.526,E2 16373.526} C_VEL
LIN {X 0,Y 345.888,Z 535.699,A -85,B 0,C 180,E1 16369.333,E2 16369.333} C_VEL
LIN {X 0,Y 345.889,Z 535.699,A -85,B 0,C 180,E1 16365.263,E2 16365.263} C_VEL
LIN {X 0,Y 345.898,Z 535.705,A -85,B 0,C 180,E1 16361.11,E2 16361.11} C_VEL
LIN {X 0,Y 345.952,Z 536.085,A -85,B 0,C 180,E1 16359.883,E2 16359.883} C_VEL
LIN {X 0,Y 348,Z 541.192,A -85,B 0,C 180,E1 16357.89,E2 16357.89} C_VEL
LIN {X 0,Y 349.884,Z 545.667,A -85,B 0,C 180,E1 16356.238,E2 16356.238} C_VEL
LIN {X 0,Y 353.474,Z 554.392,A -85,B 0,C 180,E1 16353.271,E2 16353.271} C_VEL
LIN {X 0,Y 357.544,Z 566.097,A -85,B 0,C 180,E1 16349.769,E2 16349.769} C_VEL
LIN {X 0,Y 361.358,Z 578.87,A -85,B 0,C 180,E1 16346.382,E2 16346.382} C_VEL
LIN {X 0,Y 364.401,Z 591.514,A -85,B 0,C 180,E1 16343.377,E2 16343.377} C_VEL
LIN {X 0,Y 359.944,Z 618.128,A -85,B 0,C 180,E1 16338.824,E2 16338.824} C_VEL
LIN {X 0,Y 358.384,Z 628.855,A -85,B 0,C 180,E1 16337.017,E2 16337.017} C_VEL
LIN {X 0,Y 359.365,Z 634.222,A -85,B 0,C 180,E1 16336.698,E2 16336.698} C_VEL
LIN {X 0,Y 364.802,Z 662.285,A -85,B 0,C 180,E1 16335.398,E2 16335.398} C_VEL
LIN {X 0,Y 365.316,Z 667.164,A -85,B 0,C 180,E1 16335.225,E2 16335.225} C_VEL
LIN {X 0,Y 362.228,Z 758.925,A -85,B 0,C 180,E1 16333.213,E2 16333.213} C_VEL
LIN {X 0,Y 361.393,Z 774.857,A -85,B 0,C 180,E1 16332.578,E2 16332.578} C_VEL
LIN {X 0,Y 360.157,Z 789.963,A -85,B 0,C 180,E1 16331.686,E2 16331.686} C_VEL
LIN {X 0,Y 358.524,Z 804.323,A -85,B 0,C 180,E1 16330.519,E2 16330.519} C_VEL
LIN {X 0,Y 356.639,Z 817.713,A -85,B 0,C 180,E1 16329.103,E2 16329.103} C_VEL
LIN {X 0,Y 354.638,Z 829.896,A -85,B 0,C 180,E1 16327.444,E2 16327.444} C_VEL
LIN {X 0,Y 352.818,Z 840.021,A -85,B 0,C 180,E1 16325.711,E2 16325.711} C_VEL
LIN {X 0,Y 350.863,Z 849.896,A -85,B 0,C 180,E1 16323.557,E2 16323.557} C_VEL
LIN {X 0,Y 349.271,Z 857.591,A -85,B 0,C 180,E1 16321.395,E2 16321.395} C_VEL
LIN {X 0,Y 347.855,Z 864.268,A -85,B 0,C 180,E1 16318.869,E2 16318.869} C_VEL
LIN {X 0,Y 346.87,Z 868.877,A -85,B 0,C 180,E1 16316.349,E2 16316.349} C_VEL
LIN {X 0,Y 346.21,Z 871.823,A -85,B 0,C 180,E1 16313.663,E2 16313.663} C_VEL
LIN {X 0,Y 345.87,Z 872.834,A -85,B 0,C 180,E1 16310.972,E2 16310.972} C_VEL
LIN {X 0,Y 345.815,Z 872.112,A -85,B 0,C 180,E1 16308.366,E2 16308.366} C_VEL
LIN {X 0,Y 346.017,Z 869.58,A -85,B 0,C 180,E1 16305.757,E2 16305.757} C_VEL
LIN {X 0,Y 346.468,Z 865.617,A -85,B 0,C 180,E1 16303.345,E2 16303.345} C_VEL
LIN {X 0,Y 347.261,Z 859.399,A -85,B 0,C 180,E1 16300.784,E2 16300.784} C_VEL
LIN {X 0,Y 348.276,Z 852.214,A -85,B 0,C 180,E1 16298.583,E2 16298.583} C_VEL
LIN {X 0,Y 349.601,Z 842.934,A -85,B 0,C 180,E1 16296.402,E2 16296.402} C_VEL
LIN {X 0,Y 351.035,Z 832.652,A -85,B 0,C 180,E1 16294.498,E2 16294.498} C_VEL
LIN {X 0,Y 352.636,Z 820.174,A -85,B 0,C 180,E1 16292.679,E2 16292.679} C_VEL
LIN {X 0,Y 354.114,Z 807.321,A -85,B 0,C 180,E1 16291.219,E2 16291.219} C_VEL
LIN {X 0,Y 355.454,Z 793.524,A -85,B 0,C 180,E1 16289.998,E2 16289.998} C_VEL
LIN {X 0,Y 356.541,Z 778.88,A -85,B 0,C 180,E1 16289.034,E2 16289.034} C_VEL
LIN {X 0,Y 357.353,Z 763.035,A -85,B 0,C 180,E1 16288.305,E2 16288.305} C_VEL
LIN {X 0,Y 357.893,Z 742.174,A -85,B 0,C 180,E1 16287.762,E2 16287.762} C_VEL
LIN {X 0,Y 359.789,Z 662.573,A -85,B 0,C 180,E1 16286.091,E2 16286.091} C_VEL
LIN {X 0,Y 357.953,Z 651.42,A -85,B 0,C 180,E1 16285.7,E2 16285.7} C_VEL
LIN {X 0,Y 356.218,Z 646.714,A -85,B 0,C 180,E1 16285.459,E2 16285.459} C_VEL
LIN {X 0,Y 348.637,Z 635.603,A -85,B 0,C 180,E1 16284.594,E2 16284.594} C_VEL
LIN {X 0,Y 347.243,Z 631.526,A -85,B 0,C 180,E1 16284.385,E2 16284.385} C_VEL
LIN {X 0,Y 346.914,Z 629.018,A -85,B 0,C 180,E1 16284.25,E2 16284.25} C_VEL
LIN {X 0,Y 350.445,Z 601.257,A -85,B 0,C 180,E1 16279.644,E2 16279.644} C_VEL
LIN {X 0,Y 352.415,Z 585.893,A -85,B 0,C 180,E1 16277.047,E2 16277.047} C_VEL
LIN {X 0,Y 348.177,Z 569.293,A -85,B 0,C 180,E1 16273.482,E2 16273.482} C_VEL
LIN {X 0,Y 343.526,Z 553.565,A -85,B 0,C 180,E1 16269.824,E2 16269.824} C_VEL
LIN {X 0,Y 338.684,Z 539.242,A -85,B 0,C 180,E1 16266.232,E2 16266.232} C_VEL
LIN {X 0,Y 337.956,Z 536.817,A -85,B 0,C 180,E1 16265.531,E2 16265.531} C_VEL
LIN {X 0,Y 337.953,Z 536.644,A -85,B 0,C 180,E1 16261.133,E2 16261.133} C_VEL
LIN {X 0,Y 337.947,Z 536.671,A -85,B 0,C 180,E1 16256.816,E2 16256.816} C_VEL
LIN {X 0,Y 337.95,Z 536.68,A -85,B 0,C 180,E1 16252.663,E2 16252.663} C_VEL
LIN {X 0,Y 337.952,Z 536.681,A -85,B 0,C 180,E1 16248.463,E2 16248.463} C_VEL
LIN {X 0,Y 337.948,Z 536.702,A -85,B 0,C 180,E1 16244.278,E2 16244.278} C_VEL
LIN {X 0,Y 337.94,Z 536.677,A -85,B 0,C 180,E1 16239.98,E2 16239.98} C_VEL
LIN {X 0,Y 337.943,Z 536.686,A -85,B 0,C 180,E1 16235.842,E2 16235.842} C_VEL
LIN {X 0,Y 337.94,Z 536.693,A -85,B 0,C 180,E1 16231.563,E2 16231.563} C_VEL
LIN {X 0,Y 337.938,Z 536.672,A -85,B 0,C 180,E1 16227.43,E2 16227.43} C_VEL
LIN {X 0,Y 337.936,Z 536.698,A -85,B 0,C 180,E1 16223.174,E2 16223.174} C_VEL
LIN {X 0,Y 337.936,Z 536.67,A -85,B 0,C 180,E1 16218.994,E2 16218.994} C_VEL
LIN {X 0,Y 337.933,Z 536.695,A -85,B 0,C 180,E1 16214.656,E2 16214.656} C_VEL
LIN {X 0,Y 337.935,Z 536.67,A -85,B 0,C 180,E1 16210.398,E2 16210.398} C_VEL
LIN {X 0,Y 337.941,Z 536.689,A -85,B 0,C 180,E1 16206.115,E2 16206.115} C_VEL
LIN {X 0,Y 337.943,Z 536.669,A -85,B 0,C 180,E1 16201.865,E2 16201.865} C_VEL
LIN {X 0,Y 337.953,Z 536.691,A -85,B 0,C 180,E1 16197.626,E2 16197.626} C_VEL
LIN {X 0,Y 337.959,Z 536.667,A -85,B 0,C 180,E1 16193.375,E2 16193.375} C_VEL
LIN {X 0,Y 337.972,Z 536.698,A -85,B 0,C 180,E1 16189.086,E2 16189.086} C_VEL
LIN {X 0,Y 337.989,Z 536.666,A -85,B 0,C 180,E1 16184.735,E2 16184.735} C_VEL
LIN {X 0,Y 337.983,Z 536.685,A -85,B 0,C 180,E1 16180.471,E2 16180.471} C_VEL
LIN {X 0,Y 337.986,Z 536.699,A -85,B 0,C 180,E1 16176.277,E2 16176.277} C_VEL
LIN {X 0,Y 337.975,Z 536.688,A -85,B 0,C 180,E1 16171.941,E2 16171.941} C_VEL
LIN {X 0,Y 337.973,Z 536.684,A -85,B 0,C 180,E1 16167.786,E2 16167.786} C_VEL
LIN {X 0,Y 337.967,Z 536.69,A -85,B 0,C 180,E1 16163.513,E2 16163.513} C_VEL
LIN {X 0,Y 338.023,Z 536.892,A -85,B 0,C 180,E1 16159.74,E2 16159.74} C_VEL
LIN {X 0,Y 344.475,Z 553.748,A -85,B 0,C 180,E1 16156.039,E2 16156.039} C_VEL
LIN {X 0,Y 350.73,Z 571.257,A -85,B 0,C 180,E1 16152.65,E2 16152.65} C_VEL
LIN {X 0,Y 357.098,Z 590.7,A -85,B 0,C 180,E1 16149.255,E2 16149.255} C_VEL
LIN {X 0,Y 358.151,Z 594.894,A -85,B 0,C 180,E1 16148.585,E2 16148.585} C_VEL
LIN {X 0,Y 354.611,Z 618.417,A -85,B 0,C 180,E1 16145.851,E2 16145.851} C_VEL
LIN {X 0,Y 357.487,Z 649.676,A -85,B 0,C 180,E1 16144.914,E2 16144.914} C_VEL
LIN {X 0,Y 353.455,Z 810.3,A -85,B 0,C 180,E1 16141.716,E2 16141.716} C_VEL
LIN {X 0,Y 352.261,Z 828.807,A -85,B 0,C 180,E1 16141.067,E2 16141.067} C_VEL
LIN {X 0,Y 350.527,Z 846.924,A -85,B 0,C 180,E1 16140.134,E2 16140.134} C_VEL
LIN {X 0,Y 348.526,Z 864.419,A -85,B 0,C 180,E1 16138.907,E2 16138.907} C_VEL
LIN {X 0,Y 346.388,Z 880.941,A -85,B 0,C 180,E1 16137.413,E2 16137.413} C_VEL
LIN {X 0,Y 344.161,Z 896.538,A -85,B 0,C 180,E1 16135.65,E2 16135.65} C_VEL
LIN {X 0,Y 342.067,Z 911.154,A -85,B 0,C 180,E1 16133.606,E2 16133.606} C_VEL
LIN {X 0,Y 340.175,Z 924.662,A -85,B 0,C 180,E1 16131.293,E2 16131.293} C_VEL
LIN {X 0,Y 338.635,Z 936.711,A -85,B 0,C 180,E1 16128.774,E2 16128.774} C_VEL
LIN {X 0,Y 337.535,Z 947.543,A -85,B 0,C 180,E1 16125.992,E2 16125.992} C_VEL
LIN {X 0,Y 336.957,Z 956.229,A -85,B 0,C 180,E1 16123.209,E2 16123.209} C_VEL
LIN {X 0,Y 336.819,Z 963.438,A -85,B 0,C 180,E1 16120.261,E2 16120.261} C_VEL
LIN {X 0,Y 336.987,Z 968.761,A -85,B 0,C 180,E1 16117.331,E2 16117.331} C_VEL
LIN {X 0,Y 337.305,Z 972.321,A -85,B 0,C 180,E1 16114.422,E2 16114.422} C_VEL
LIN {X 0,Y 337.532,Z 974.112,A -85,B 0,C 180,E1 16111.699,E2 16111.699} C_VEL
LIN {X 0,Y 337.543,Z 974.437,A -85,B 0,C 180,E1 16108.984,E2 16108.984} C_VEL
LIN {X 0,Y 337.306,Z 973.178,A -85,B 0,C 180,E1 16106.093,E2 16106.093} C_VEL
LIN {X 0,Y 336.954,Z 970.278,A -85,B 0,C 180,E1 16103.186,E2 16103.186} C_VEL
LIN {X 0,Y 336.729,Z 965.712,A -85,B 0,C 180,E1 16100.259,E2 16100.259} C_VEL
LIN {X 0,Y 336.8,Z 959.411,A -85,B 0,C 180,E1 16097.313,E2 16097.313} C_VEL
LIN {X 0,Y 337.379,Z 951.239,A -85,B 0,C 180,E1 16094.358,E2 16094.358} C_VEL
LIN {X 0,Y 338.559,Z 940.958,A -85,B 0,C 180,E1 16091.404,E2 16091.404} C_VEL
LIN {X 0,Y 340.212,Z 929.837,A -85,B 0,C 180,E1 16088.812,E2 16088.812} C_VEL
LIN {X 0,Y 342.299,Z 917.328,A -85,B 0,C 180,E1 16086.415,E2 16086.415} C_VEL
LIN {X 0,Y 344.727,Z 903.359,A -85,B 0,C 180,E1 16084.215,E2 16084.215} C_VEL
LIN {X 0,Y 347.497,Z 887.759,A -85,B 0,C 180,E1 16082.222,E2 16082.222} C_VEL
LIN {X 0,Y 350.117,Z 871.674,A -85,B 0,C 180,E1 16080.576,E2 16080.576} C_VEL
LIN {X 0,Y 352.61,Z 854.874,A -85,B 0,C 180,E1 16079.225,E2 16079.225} C_VEL
LIN {X 0,Y 354.813,Z 837.421,A -85,B 0,C 180,E1 16078.157,E2 16078.157} C_VEL
LIN {X 0,Y 356.642,Z 818.919,A -85,B 0,C 180,E1 16077.356,E2 16077.356} C_VEL
LIN {X 0,Y 357.672,Z 800.445,A -85,B 0,C 180,E1 16076.839,E2 16076.839} C_VEL
LIN {X 0,Y 362.113,Z 647.429,A -85,B 0,C 180,E1 16073.732,E2 16073.732} C_VEL
LIN {X 0,Y 359.153,Z 619.411,A -85,B 0,C 180,E1 16072.697,E2 16072.697} C_VEL
LIN {X 0,Y 360.569,Z 610.888,A -85,B 0,C 180,E1 16071.698,E2 16071.698} C_VEL
LIN {X 0,Y 362.665,Z 599.504,A -85,B 0,C 180,E1 16070.281,E2 16070.281} C_VEL
LIN {X 0,Y 358.294,Z 585.369,A -85,B 0,C 180,E1 16067.453,E2 16067.453} C_VEL
LIN {X 0,Y 353.297,Z 571.575,A -85,B 0,C 180,E1 16064.282,E2 16064.282} C_VEL
LIN {X 0,Y 348.649,Z 560.314,A -85,B 0,C 180,E1 16061.269,E2 16061.269} C_VEL
LIN {X 0,Y 345.2,Z 552.655,A -85,B 0,C 180,E1 16058.942,E2 16058.942} C_VEL
LIN {X 0,Y 342.965,Z 547.833,A -85,B 0,C 180,E1 16057.329,E2 16057.329} C_VEL
LIN {X 0,Y 341.557,Z 544.769,A -85,B 0,C 180,E1 16056.251,E2 16056.251} C_VEL
LIN {X 0,Y 339.492,Z 540.509,A -85,B 0,C 180,E1 16054.64,E2 16054.64} C_VEL
LIN {X 0,Y 337.963,Z 536.847,A -85,B 0,C 180,E1 16053.11,E2 16053.11} C_VEL
LIN {X 0,Y 337.935,Z 536.687,A -85,B 0,C 180,E1 16048.834,E2 16048.834} C_VEL
LIN {X 0,Y 337.93,Z 536.686,A -85,B 0,C 180,E1 16044.657,E2 16044.657} C_VEL
LIN {X 0,Y 337.926,Z 536.689,A -85,B 0,C 180,E1 16040.434,E2 16040.434} C_VEL
LIN {X 0,Y 337.926,Z 536.696,A -85,B 0,C 180,E1 16036.148,E2 16036.148} C_VEL
LIN {X 0,Y 337.926,Z 536.705,A -85,B 0,C 180,E1 16031.953,E2 16031.953} C_VEL
LIN {X 0,Y 337.937,Z 536.698,A -85,B 0,C 180,E1 16027.651,E2 16027.651} C_VEL
LIN {X 0,Y 337.948,Z 536.682,A -85,B 0,C 180,E1 16023.392,E2 16023.392} C_VEL
